C01810=1088.050,222.175,424.742,176.092,21.360,153.325
C01811=1088.041,221.787,424.782,176.088,21.356,153.325
C01812=1088.035,221.538,424.807,176.086,21.354,153.325
C01813=1088.029,221.290,424.832,176.082,21.351,153.325
C01814=1088.024,221.041,424.857,176.080,21.349,153.324
C01815=1088.018,220.792,424.883,176.077,21.347,153.324
C01816=1088.012,220.544,424.908,176.075,21.344,153.324
C01817=1088.007,220.295,424.932,176.072,21.341,153.324
C01818=1088.000,220.046,424.958,176.069,21.339,153.324
C01819=1087.995,219.798,424.983,176.066,21.336,153.324
C01820=1087.990,219.549,425.008,176.064,21.334,153.324
C01821=1087.984,219.301,425.033,176.061,21.332,153.324
C01822=1087.978,219.051,425.057,176.058,21.329,153.324
C01823=1087.973,218.803,425.083,176.055,21.327,153.324
C01824=1087.967,218.554,425.108,176.053,21.325,153.323
C01825=1087.961,218.305,425.133,176.050,21.322,153.323
C01826=1087.955,218.057,425.158,176.048,21.320,153.323
C01827=1087.950,217.808,425.182,176.044,21.317,153.323
C01828=1087.945,217.560,425.208,176.042,21.314,153.323
C01829=1087.939,217.310,425.233,176.039,21.312,153.323
C01830=1087.934,217.062,425.257,176.037,21.310,153.323
C01831=1087.927,216.813,425.282,176.035,21.307,153.323
C01832=1087.922,216.564,425.307,176.031,21.305,153.323
C01833=1087.917,216.315,425.332,176.029,21.303,153.322
C01834=1087.911,216.067,425.357,176.026,21.300,153.322
C01835=1087.905,215.818,425.382,176.024,21.298,153.322
C01836=1087.900,215.570,425.406,176.021,21.295,153.322
C01837=1087.894,215.320,425.431,176.018,21.292,153.322
C01838=1087.888,215.072,425.456,176.015,21.290,153.322
C01839=1087.883,214.824,425.480,176.013,21.288,153.322
C01840=1087.877,214.575,425.506,176.010,21.285,153.322
C01841=1087.872,214.326,425.530,176.008,21.283,153.322
C01842=1087.866,214.077,425.555,176.005,21.280,153.322
C01843=1087.861,213.829,425.580,176.002,21.278,153.321
C01844=1087.855,213.580,425.605,175.999,21.275,153.321
C01845=1087.849,213.331,425.629,175.997,21.273,153.321
C01846=1087.844,213.082,425.653,175.995,21.270,153.321
C01847=1087.838,212.834,425.678,175.991,21.268,153.321
C01848=1087.833,212.585,425.703,175.989,21.266,153.321
C01849=1087.827,212.336,425.727,175.986,21.263,153.321
C01850=1087.821,212.087,425.752,175.984,21.261,153.321
C01851=1087.815,211.839,425.777,175.981,21.258,153.321
C01852=1087.810,211.590,425.801,175.978,21.256,153.321
C01853=1087.805,211.341,425.825,175.975,21.253,153.320
C01854=1087.799,211.092,425.850,175.973,21.251,153.320
C01855=1087.793,210.844,425.874,175.970,21.248,153.320
C01856=1087.787,210.595,425.900,175.968,21.246,153.320
C01857=1087.782,210.346,425.924,175.965,21.244,153.320
C01858=1087.777,210.098,425.948,175.962,21.241,153.320
C01859=1087.771,209.848,425.973,175.960,21.239,153.320
C01860=1087.762,209.464,426.010,175.955,21.235,153.320
C01861=1087.754,209.080,426.048,175.952,21.231,153.319
C01862=1087.745,208.695,426.086,175.948,21.228,153.319
C01863=1087.736,208.311,426.123,175.944,21.224,153.319
C01864=1087.713,207.286,426.222,175.868,21.185,153.323
C01865=1087.707,207.037,426.246,175.866,21.184,153.323
C01866=1087.702,206.788,426.269,175.863,21.182,153.323
C01867=1087.696,206.539,426.293,175.860,21.181,153.323
C01868=1087.690,206.291,426.318,175.857,21.179,153.323
C01869=1087.685,206.042,426.342,175.855,21.178,153.323
C01870=1087.679,205.793,426.365,175.852,21.176,153.323
C01871=1087.674,205.545,426.389,175.849,21.175,153.324
C01872=1087.669,205.296,426.413,175.846,21.173,153.324
C01873=1087.662,205.046,426.437,175.843,21.172,153.324
C01874=1087.657,204.798,426.461,175.841,21.170,153.324
C01875=1087.651,204.549,426.484,175.838,21.169,153.324
C01876=1087.646,204.300,426.508,175.836,21.167,153.324
C01877=1087.641,204.052,426.532,175.833,21.166,153.324
C01878=1087.635,203.803,426.555,175.829,21.164,153.324
C01879=1087.630,203.554,426.580,175.827,21.163,153.325
C01880=1087.624,203.305,426.603,175.824,21.161,153.325
C01881=1087.618,203.056,426.627,175.822,21.159,153.325
C01882=1087.613,202.807,426.651,175.819,21.158,153.325
C01883=1087.607,202.559,426.674,175.817,21.156,153.325
C01884=1087.601,202.310,426.697,175.814,21.155,153.325
C01885=1087.596,202.061,426.722,175.811,21.153,153.325
C01886=1087.590,201.812,426.744,175.808,21.152,153.325
C01887=1087.585,201.564,426.769,175.805,21.151,153.325
C01888=1087.579,201.314,426.792,175.803,21.149,153.326
C01889=1087.573,201.066,426.816,175.800,21.148,153.326
C01890=1087.568,200.816,426.839,175.797,21.147,153.326
C01891=1087.562,200.568,426.863,175.795,21.145,153.326
C01892=1087.556,200.319,426.886,175.791,21.143,153.326
C01893=1087.550,200.071,426.910,175.789,21.142,153.326
C01894=1087.545,199.822,426.933,175.786,21.140,153.326
C01895=1087.539,199.573,426.956,175.784,21.139,153.326
C01896=1087.533,199.324,426.981,175.781,21.138,153.326
C01897=1087.527,199.075,427.004,175.778,21.136,153.327
C01898=1087.522,198.826,427.027,175.776,21.135,153.327
C01899=1087.516,198.577,427.051,175.773,21.133,153.327
C01900=1087.511,198.328,427.074,175.770,21.131,153.327
C01901=1087.505,198.079,427.097,175.767,21.130,153.327
C01902=1087.500,197.831,427.121,175.764,21.129,153.327
C01903=1087.494,197.582,427.144,175.762,21.127,153.327
C01904=1087.488,197.333,427.167,175.759,21.125,153.327
C01905=1087.483,197.084,427.191,175.757,21.124,153.327
C01906=1087.477,196.836,427.214,175.754,21.122,153.327
C01907=1087.471,196.587,427.237,175.752,21.121,153.328
C01908=1087.466,196.337,427.260,175.749,21.120,153.328
C01909=1087.460,196.089,427.284,175.746,21.118,153.328
C01910=1087.455,195.840,427.307,175.743,21.116,153.328
C01911=1087.449,195.591,427.330,175.740,21.115,153.328
C01912=1087.444,195.342,427.354,175.738,21.113,153.328
C01913=1087.438,195.093,427.377,175.735,21.112,153.328
C01914=1087.432,194.845,427.400,175.733,21.111,153.328
C01915=1087.426,194.596,427.423,175.730,21.109,153.329
C01916=1087.421,194.347,427.447,175.727,21.108,153.329
C01917=1087.416,194.098,427.470,175.725,21.106,153.329
C01918=1087.410,193.849,427.493,175.722,21.104,153.329
C01919=1087.404,193.600,427.516,175.720,21.103,153.329
C01920=1087.399,193.351,427.539,175.716,21.101,153.329
C01921=1087.393,193.103,427.563,175.714,21.100,153.329
C01922=1087.387,192.854,427.586,175.711,21.098,153.329
C01923=1087.382,192.605,427.609,175.709,21.097,153.329
C01924=1087.376,192.356,427.632,175.706,21.095,153.329
C01925=1087.371,192.079,427.657,175.703,21.094,153.330
C01926=1087.364,191.801,427.683,175.700,21.092,153.330
C01927=1087.358,191.523,427.709,175.697,21.090,153.330
C01928=1087.352,191.245,427.734,175.694,21.088,153.330
C01929=1087.347,190.997,427.757,175.691,21.087,153.330
C01930=1087.341,190.748,427.780,175.689,21.085,153.330
C01931=1087.336,190.499,427.804,175.686,21.084,153.330
C01932=1087.330,190.250,427.826,175.684,21.082,153.330
C01933=1087.324,190.001,427.849,175.681,21.081,153.330
C01934=1087.319,189.752,427.872,175.679,21.079,153.330
C01935=1087.313,189.503,427.895,175.676,21.078,153.331
C01936=1087.307,189.254,427.918,175.673,21.076,153.331
C01937=1087.303,189.006,427.941,175.671,21.075,153.331
C01938=1087.297,188.757,427.964,175.668,21.073,153.331
C01939=1087.291,188.508,427.987,175.666,21.072,153.331
C01940=1087.286,188.259,428.010,175.663,21.070,153.331
C01941=1087.280,188.010,428.032,175.661,21.069,153.331
C01942=1087.275,187.761,428.055,175.658,21.067,153.331
C01943=1087.269,187.513,428.078,175.656,21.066,153.331
C01944=1087.264,187.263,428.102,175.653,21.064,153.331
C01945=1087.259,187.014,428.125,175.650,21.063,153.331
C01946=1087.253,186.766,428.147,175.648,21.061,153.332
C01947=1087.248,186.517,428.169,175.645,21.059,153.332
C01948=1087.242,186.268,428.192,175.642,21.057,153.332
C01949=1087.237,186.019,428.215,175.639,21.056,153.332
C01950=1087.231,185.770,428.238,175.637,21.055,153.332
C01951=1087.226,185.522,428.261,175.634,21.053,153.332
C01952=1087.220,185.272,428.283,175.632,21.051,153.332
C01953=1087.215,185.023,428.307,175.629,21.050,153.332
C01954=1087.209,184.775,428.329,175.627,21.048,153.332
C01955=1087.203,184.525,428.351,175.624,21.047,153.332
C01956=1087.198,184.276,428.374,175.621,21.046,153.332
C01957=1087.192,184.027,428.397,175.619,21.044,153.333
C01958=1087.186,183.779,428.419,175.616,21.043,153.333
C01959=1087.181,183.530,428.441,175.614,21.041,153.333
C01960=1087.175,183.281,428.464,175.611,21.040,153.333
C01961=1087.169,183.032,428.487,175.609,21.038,153.333
C01962=1087.163,182.783,428.509,175.606,21.037,153.333
C01963=1087.157,182.534,428.532,175.603,21.035,153.333
C01964=1087.152,182.286,428.554,175.601,21.034,153.333
C01965=1087.147,182.036,428.576,175.598,21.032,153.333
C01966=1087.140,181.788,428.599,175.596,21.031,153.333
C01967=1087.135,181.538,428.621,175.593,21.030,153.334
C01968=1087.129,181.289,428.644,175.590,21.028,153.334
C01969=1087.123,181.041,428.666,175.588,21.027,153.334
C01970=1087.118,180.792,428.688,175.585,21.025,153.334
C01971=1087.112,180.543,428.711,175.583,21.024,153.334
C01972=1087.107,180.293,428.733,175.580,21.022,153.334
C01973=1087.100,180.045,428.756,175.578,21.021,153.334
C01974=1087.095,179.796,428.778,175.575,21.019,153.334
C01975=1087.090,179.547,428.801,175.572,21.018,153.334
C01976=1087.083,179.298,428.822,175.570,21.016,153.335
C01977=1087.078,179.049,428.845,175.567,21.015,153.335
C01978=1087.073,178.800,428.867,175.565,21.013,153.335
C01979=1087.066,178.552,428.889,175.562,21.012,153.335
C01980=1087.061,178.302,428.912,175.560,21.011,153.335
C01981=1087.055,178.053,428.935,175.558,21.009,153.335
C01982=1087.050,177.805,428.956,175.555,21.008,153.335
C01983=1087.044,177.555,428.978,175.553,21.006,153.335
C01984=1087.039,177.306,429.001,175.550,21.005,153.335
C01985=1087.033,177.058,429.022,175.548,21.003,153.335
C01986=1087.027,176.809,429.045,175.545,21.002,153.335
C01987=1087.021,176.560,429.067,175.543,21.000,153.335
C01988=1087.016,176.310,429.089,175.540,20.999,153.336
C01989=1087.010,176.033,429.114,175.537,20.996,153.336
C01990=1087.003,175.755,429.139,175.534,20.995,153.336
C01991=1086.997,175.476,429.164,175.531,20.994,153.336
C01992=1086.991,175.199,429.188,175.529,20.992,153.336
C01993=1086.985,174.949,429.210,175.526,20.991,153.336
C01994=1086.980,174.701,429.232,175.524,20.989,153.336
C01995=1086.974,174.452,429.254,175.521,20.987,153.336
C01996=1086.969,174.203,429.276,175.519,20.986,153.336
C01997=1086.963,173.955,429.298,175.516,20.984,153.336
C01998=1086.957,173.705,429.321,175.514,20.983,153.336
C01999=1086.952,173.456,429.343,175.511,20.981,153.337
C02000=1086.946,173.207,429.364,175.508,20.980,153.337
C02001=1086.941,172.958,429.387,175.506,20.978,153.337
C02002=1086.935,172.710,429.408,175.504,20.976,153.337
C02003=1086.930,172.460,429.430,175.501,20.975,153.337
C02004=1086.923,172.211,429.452,175.498,20.974,153.337
C02005=1086.919,171.962,429.474,175.496,20.972,153.337
C02006=1086.913,171.713,429.497,175.493,20.970,153.337
C02007=1086.907,171.465,429.518,175.491,20.969,153.337
C02008=1086.902,171.215,429.540,175.489,20.967,153.337
C02009=1086.896,170.967,429.562,175.487,20.966,153.337
C02010=1086.891,170.717,429.584,175.484,20.965,153.337
C02011=1086.885,170.468,429.606,175.482,20.963,153.337
C02012=1086.880,170.219,429.627,175.479,20.961,153.337
C02013=1086.874,169.970,429.649,175.476,20.960,153.338
C02014=1086.869,169.722,429.672,175.474,20.958,153.338
C02015=1086.862,169.473,429.693,175.471,20.956,153.338
C02016=1086.858,169.224,429.715,175.469,20.955,153.338
C02017=1086.851,168.975,429.737,175.466,20.953,153.338
C02018=1086.847,168.726,429.759,175.464,20.952,153.338
C02019=1086.840,168.477,429.780,175.461,20.950,153.338
C02020=1086.836,168.228,429.802,175.460,20.949,153.338
C02021=1086.829,167.979,429.824,175.457,20.947,153.338
C02022=1086.825,167.730,429.846,175.455,20.945,153.338
C02023=1086.818,167.481,429.867,175.452,20.944,153.338
C02024=1086.814,167.232,429.889,175.450,20.942,153.338
C02025=1086.807,166.983,429.911,175.447,20.941,153.338
C02026=1086.803,166.734,429.933,175.445,20.939,153.338
C02027=1086.796,166.485,429.954,175.442,20.937,153.338
C02028=1086.792,166.236,429.976,175.440,20.936,153.339
C02029=1086.786,165.987,429.997,175.437,20.934,153.339
C02030=1086.781,165.738,430.020,175.435,20.933,153.339
C02031=1086.775,165.489,430.041,175.433,20.931,153.339
C02032=1086.770,165.239,430.062,175.431,20.930,153.339
C02033=1086.764,164.991,430.084,175.428,20.928,153.339
C02034=1086.758,164.741,430.105,175.426,20.926,153.339
C02035=1086.753,164.493,430.127,175.423,20.925,153.339
C02036=1086.748,164.244,430.148,175.421,20.923,153.339
C02037=1086.742,163.994,430.171,175.418,20.921,153.339
C02038=1086.737,163.746,430.192,175.416,20.920,153.339
C02039=1086.732,163.496,430.213,175.413,20.918,153.339
C02040=1086.726,163.247,430.235,175.411,20.917,153.339
C02041=1086.721,162.999,430.256,175.409,20.915,153.339
C02042=1086.715,162.749,430.278,175.406,20.914,153.339
C02043=1086.710,162.501,430.300,175.404,20.912,153.339
C02044=1086.705,162.251,430.321,175.402,20.910,153.339
C02045=1086.699,162.002,430.342,175.399,20.908,153.339
C02046=1086.693,161.754,430.364,175.397,20.907,153.339
C02047=1086.689,161.505,430.385,175.394,20.905,153.339
C02048=1086.683,161.255,430.406,175.392,20.904,153.339
C02049=1086.677,161.007,430.428,175.390,20.903,153.340
C02050=1086.671,160.757,430.449,175.387,20.901,153.340
C02051=1086.665,160.509,430.471,175.385,20.899,153.340
C02052=1086.660,160.259,430.492,175.382,20.897,153.340
C02053=1086.654,159.981,430.516,175.380,20.896,153.340
C02054=1086.647,159.703,430.539,175.377,20.894,153.340
C02055=1086.642,159.424,430.563,175.375,20.893,153.340
C02056=1086.635,159.146,430.587,175.372,20.890,153.340
C02057=1086.630,158.897,430.608,175.370,20.889,153.340
C02058=1086.623,158.648,430.629,175.367,20.888,153.340
C02059=1086.618,158.399,430.650,175.365,20.886,153.340
C02060=1086.613,158.150,430.672,175.362,20.884,153.340
C02061=1086.607,157.901,430.694,175.360,20.883,153.340
C02062=1086.602,157.652,430.714,175.357,20.881,153.340
C02063=1086.596,157.403,430.735,175.355,20.879,153.340
C02064=1086.590,157.153,430.756,175.353,20.878,153.340
C02065=1086.585,156.905,430.778,175.351,20.876,153.340
C02066=1086.580,156.656,430.798,175.348,20.875,153.341
C02067=1086.573,156.407,430.820,175.346,20.873,153.341
C02068=1086.568,156.158,430.841,175.343,20.872,153.341
C02069=1086.563,155.909,430.862,175.341,20.870,153.341
C02070=1086.556,155.660,430.883,175.339,20.869,153.341
C02071=1086.551,155.411,430.904,175.337,20.867,153.341
C02072=1086.546,155.162,430.925,175.334,20.865,153.341
C02073=1086.540,154.912,430.946,175.332,20.863,153.341
C02074=1086.534,154.664,430.967,175.329,20.862,153.341
C02075=1086.529,154.415,430.988,175.327,20.861,153.341
C02076=1086.523,154.165,431.009,175.325,20.859,153.341
C02077=1086.518,153.916,431.030,175.323,20.858,153.341
C02078=1086.512,153.667,431.051,175.320,20.856,153.341
C02079=1086.506,153.418,431.072,175.318,20.854,153.341
C02080=1086.501,153.169,431.093,175.315,20.852,153.341
C02081=1086.495,152.920,431.114,175.314,20.851,153.341
C02082=1086.489,152.670,431.135,175.311,20.850,153.341
C02083=1086.484,152.421,431.155,175.309,20.848,153.341
C02084=1086.479,152.173,431.177,175.306,20.846,153.341
C02085=1086.473,151.924,431.197,175.304,20.844,153.341
C02086=1086.468,151.674,431.218,175.302,20.843,153.341
C02087=1086.462,151.425,431.239,175.300,20.841,153.341
C02088=1086.457,151.176,431.260,175.297,20.840,153.342
C02089=1086.451,150.927,431.281,175.295,20.838,153.342
C02090=1086.445,150.678,431.302,175.292,20.837,153.342
C02091=1086.439,150.429,431.322,175.290,20.835,153.342
C02092=1086.434,150.180,431.343,175.288,20.833,153.342
C02093=1086.429,149.932,431.364,175.286,20.832,153.342
C02094=1086.423,149.682,431.385,175.283,20.830,153.342
C02095=1086.417,149.433,431.405,175.281,20.829,153.342
C02096=1086.412,149.183,431.426,175.278,20.827,153.342
C02097=1086.406,148.935,431.447,175.277,20.825,153.342
C02098=1086.401,148.686,431.467,175.274,20.824,153.342
C02099=1086.395,148.436,431.488,175.272,20.822,153.342
C02100=1086.389,148.187,431.509,175.269,20.820,153.342
C02101=1086.384,147.939,431.530,175.268,20.819,153.342
C02102=1086.378,147.690,431.550,175.265,20.818,153.342
C02103=1086.372,147.440,431.571,175.263,20.816,153.342
C02104=1086.367,147.191,431.591,175.260,20.814,153.342
C02105=1086.362,146.942,431.612,175.258,20.812,153.342
C02106=1086.355,146.694,431.633,175.256,20.811,153.342
C02107=1086.350,146.444,431.653,175.253,20.809,153.342
C02108=1086.344,146.195,431.674,175.251,20.807,153.342
C02109=1086.339,145.946,431.695,175.249,20.806,153.342
C02110=1086.333,145.697,431.715,175.247,20.805,153.342
C02111=1086.328,145.448,431.735,175.245,20.803,153.342
C02112=1086.322,145.198,431.756,175.242,20.801,153.342
C02113=1086.316,144.949,431.776,175.240,20.799,153.342
C02114=1086.311,144.700,431.797,175.237,20.797,153.342
C02115=1086.305,144.451,431.817,175.236,20.796,153.342
C02116=1086.299,144.203,431.838,175.233,20.795,153.342
C02117=1086.293,143.924,431.860,175.231,20.793,153.342
C02118=1086.286,143.645,431.884,175.228,20.791,153.343
C02119=1086.281,143.367,431.906,175.226,20.789,153.343
C02120=1086.274,143.087,431.929,175.223,20.787,153.343
C02121=1086.269,142.838,431.949,175.221,20.786,153.343
C02122=1086.263,142.589,431.969,175.218,20.784,153.343
C02123=1086.258,142.340,431.990,175.216,20.782,153.343
C02124=1086.252,142.091,432.011,175.214,20.781,153.343
C02125=1086.246,141.842,432.031,175.212,20.779,153.343
C02126=1086.241,141.593,432.051,175.210,20.777,153.343
C02127=1086.236,141.344,432.072,175.207,20.775,153.343
C02128=1086.230,141.095,432.092,175.205,20.774,153.343
C02129=1086.225,140.846,432.112,175.203,20.772,153.343
C02130=1086.219,140.596,432.133,175.201,20.771,153.343
C02131=1086.213,140.347,432.153,175.198,20.769,153.343
C02132=1086.208,140.098,432.174,175.197,20.768,153.343
C02133=1086.202,139.850,432.194,175.194,20.766,153.343
C02134=1086.196,139.600,432.214,175.192,20.764,153.343
C02135=1086.190,139.352,432.234,175.189,20.762,153.343
C02136=1086.185,139.102,432.254,175.188,20.761,153.343
C02137=1086.179,138.853,432.274,175.185,20.759,153.343
C02138=1086.174,138.604,432.294,175.183,20.758,153.343
C02139=1086.168,138.355,432.314,175.180,20.756,153.343
C02140=1086.163,138.106,432.335,175.179,20.754,153.343
C02141=1086.157,137.857,432.355,175.176,20.753,153.343
C02142=1086.151,137.607,432.375,175.174,20.751,153.343
C02143=1086.145,137.358,432.395,175.172,20.749,153.343
C02144=1086.140,137.109,432.416,175.170,20.747,153.343
C02145=1086.134,136.860,432.436,175.167,20.746,153.343
C02146=1086.128,136.611,432.455,175.165,20.744,153.343
C02147=1086.123,136.361,432.475,175.163,20.742,153.343
C02148=1086.117,136.113,432.495,175.161,20.741,153.343
C02149=1086.112,135.863,432.516,175.159,20.739,153.343
C02150=1086.106,135.614,432.535,175.156,20.737,153.343
C02151=1086.101,135.365,432.556,175.155,20.736,153.343
C02152=1086.095,135.116,432.576,175.152,20.734,153.343
C02153=1086.089,134.867,432.596,175.150,20.733,153.343
C02154=1086.084,134.618,432.615,175.147,20.731,153.343
C02155=1086.078,134.369,432.635,175.146,20.729,153.343
C02156=1086.073,134.120,432.656,175.143,20.727,153.343
C02157=1086.067,133.870,432.675,175.141,20.725,153.343
C02158=1086.061,133.621,432.695,175.139,20.724,153.343
C02159=1086.056,133.372,432.716,175.137,20.722,153.343
C02160=1086.050,133.123,432.735,175.135,20.721,153.343
C02161=1086.045,132.874,432.755,175.132,20.719,153.343
C02162=1086.039,132.624,432.775,175.131,20.717,153.343
C02163=1086.033,132.375,432.795,175.128,20.716,153.343
C02164=1086.028,132.126,432.815,175.126,20.714,153.343
C02165=1086.022,131.877,432.834,175.124,20.712,153.343
C02166=1086.016,131.628,432.854,175.122,20.710,153.343
C02167=1086.011,131.379,432.874,175.119,20.709,153.343
C02168=1086.005,131.130,432.894,175.118,20.708,153.343
C02169=1086.000,130.880,432.913,175.115,20.706,153.343
C02170=1085.994,130.631,432.933,175.113,20.704,153.343
C02171=1085.988,130.382,432.953,175.110,20.702,153.343
C02172=1085.982,130.133,432.973,175.109,20.701,153.343
C02173=1085.976,129.884,432.992,175.107,20.699,153.343
C02174=1085.970,129.635,433.012,175.104,20.697,153.343
C02175=1085.965,129.385,433.032,175.103,20.695,153.343
C02176=1085.959,129.136,433.052,175.100,20.694,153.343
C02177=1085.954,128.887,433.071,175.098,20.692,153.343
C02178=1085.948,128.638,433.091,175.096,20.691,153.343
C02179=1085.942,128.389,433.110,175.094,20.689,153.343
C02180=1085.937,128.140,433.130,175.091,20.687,153.343
C02181=1085.930,127.861,433.152,175.089,20.685,153.343
C02182=1085.924,127.582,433.174,175.087,20.683,153.343
C02183=1085.917,127.304,433.195,175.084,20.682,153.343
C02184=1085.912,127.025,433.218,175.082,20.680,153.343
C02185=1085.906,126.776,433.237,175.080,20.678,153.343
C02186=1085.900,126.527,433.257,175.078,20.676,153.343
C02187=1085.894,126.278,433.276,175.075,20.674,153.343
C02188=1085.889,126.028,433.295,175.074,20.673,153.343
C02189=1085.883,125.779,433.315,175.072,20.671,153.343
C02190=1085.877,125.530,433.335,175.069,20.669,153.343
C02191=1085.872,125.281,433.354,175.068,20.668,153.343
C02192=1085.866,125.032,433.374,175.065,20.666,153.343
C02193=1085.861,124.783,433.393,175.063,20.664,153.343
C02194=1085.855,124.533,433.413,175.061,20.663,153.343
C02195=1085.849,124.284,433.433,175.059,20.661,153.343
C02196=1085.843,124.035,433.452,175.056,20.659,153.343
C02197=1085.838,123.786,433.471,175.055,20.657,153.343
C02198=1085.833,123.537,433.490,175.053,20.655,153.343
C02199=1085.827,123.288,433.510,175.050,20.654,153.343
C02200=1085.821,123.039,433.529,175.049,20.652,153.343
C02201=1085.815,122.789,433.548,175.046,20.650,153.343
C02202=1085.810,122.540,433.568,175.044,20.648,153.343
C02203=1085.804,122.291,433.588,175.042,20.647,153.343
C02204=1085.799,122.042,433.606,175.040,20.645,153.343
C02205=1085.793,121.793,433.626,175.038,20.643,153.343
C02206=1085.787,121.543,433.645,175.036,20.641,153.343
C02207=1085.781,121.294,433.664,175.034,20.639,153.343
C02208=1085.775,121.045,433.684,175.031,20.638,153.343
C02209=1085.771,120.796,433.704,175.030,20.636,153.343
C02210=1085.765,120.547,433.723,175.028,20.634,153.343
C02211=1085.760,120.297,433.742,175.025,20.632,153.343
C02212=1085.754,120.048,433.761,175.024,20.631,153.343
C02213=1085.748,119.798,433.781,175.021,20.629,153.343
C02214=1085.743,119.550,433.799,175.019,20.627,153.343
C02215=1085.737,119.301,433.819,175.017,20.625,153.343
C02216=1085.732,119.051,433.839,175.015,20.624,153.343
C02217=1085.726,118.802,433.858,175.014,20.622,153.343
C02218=1085.721,118.553,433.877,175.011,20.620,153.343
C02219=1085.715,118.304,433.896,175.009,20.618,153.343
C02220=1085.709,118.054,433.915,175.007,20.617,153.343
C02221=1085.704,117.806,433.934,175.005,20.615,153.343
C02222=1085.699,117.556,433.953,175.003,20.613,153.343
C02223=1085.693,117.307,433.973,175.001,20.611,153.343
C02224=1085.687,117.057,433.992,174.999,20.609,153.343
C02225=1085.681,116.809,434.010,174.996,20.608,153.343
C02226=1085.676,116.559,434.029,174.995,20.606,153.342
C02227=1085.670,116.310,434.049,174.993,20.604,153.342
C02228=1085.665,116.061,434.067,174.991,20.602,153.342
C02229=1085.659,115.812,434.087,174.989,20.600,153.342
C02230=1085.654,115.562,434.106,174.986,20.598,153.342
C02231=1085.649,115.314,434.125,174.985,20.597,153.342
C02232=1085.643,115.064,434.144,174.983,20.595,153.342
C02233=1085.637,114.815,434.163,174.980,20.593,153.342
C02234=1085.632,114.566,434.182,174.979,20.591,153.342
C02235=1085.626,114.317,434.201,174.977,20.589,153.342
C02236=1085.621,114.067,434.221,174.975,20.588,153.342
C02237=1085.614,113.818,434.239,174.973,20.586,153.342
C02238=1085.609,113.569,434.258,174.970,20.584,153.342
C02239=1085.604,113.319,434.277,174.969,20.582,153.342
C02240=1085.598,113.070,434.296,174.966,20.580,153.342
C02241=1085.593,112.821,434.315,174.964,20.578,153.342
C02242=1085.587,112.572,434.334,174.963,20.577,153.342
C02243=1085.581,112.323,434.353,174.960,20.575,153.342
C02244=1085.576,112.074,434.372,174.959,20.574,153.342
C02245=1085.570,111.795,434.393,174.957,20.571,153.342
C02246=1085.563,111.516,434.414,174.954,20.569,153.342
C02247=1085.556,111.237,434.434,174.952,20.567,153.342
C02248=1085.550,110.958,434.455,174.949,20.565,153.342
C02249=1085.545,110.710,434.474,174.947,20.563,153.342
C02250=1085.539,110.461,434.493,174.946,20.561,153.342
C02251=1085.533,110.211,434.512,174.943,20.559,153.342
C02252=1085.528,109.961,434.531,174.942,20.558,153.341
C02253=1085.522,109.713,434.549,174.940,20.556,153.341
C02254=1085.516,109.463,434.568,174.937,20.554,153.341
C02255=1085.511,109.215,434.587,174.936,20.553,153.341
C02256=1085.505,108.965,434.605,174.933,20.551,153.341
C02257=1085.499,108.715,434.624,174.932,20.549,153.341
C02258=1085.493,108.467,434.643,174.929,20.547,153.341
C02259=1085.488,108.217,434.661,174.927,20.545,153.341
C02260=1085.482,107.967,434.680,174.926,20.543,153.341
C02261=1085.476,107.719,434.699,174.923,20.541,153.341
C02262=1085.471,107.469,434.717,174.922,20.540,153.341
C02263=1085.465,107.220,434.736,174.919,20.538,153.341
C02264=1085.460,106.971,434.755,174.917,20.536,153.341
C02265=1085.454,106.721,434.773,174.916,20.534,153.341
C02266=1085.448,106.473,434.792,174.913,20.532,153.341
C02267=1085.443,106.223,434.811,174.912,20.531,153.341
C02268=1085.436,105.973,434.829,174.910,20.529,153.341
C02269=1085.431,105.725,434.848,174.907,20.527,153.341
C02270=1085.425,105.476,434.866,174.906,20.525,153.341
C02271=1085.420,105.226,434.884,174.904,20.523,153.341
C02272=1085.415,104.977,434.904,174.902,20.522,153.341
C02273=1085.409,104.728,434.921,174.900,20.520,153.341
C02274=1085.403,104.478,434.940,174.898,20.518,153.341
C02275=1085.398,104.229,434.958,174.896,20.516,153.340
C02276=1085.392,103.980,434.977,174.894,20.514,153.340
C02277=1085.386,103.731,434.996,174.892,20.512,153.340
C02278=1085.381,103.481,435.014,174.890,20.510,153.340
C02279=1085.374,103.232,435.033,174.889,20.508,153.340
C02280=1085.370,102.983,435.051,174.886,20.506,153.340
C02281=1085.363,102.734,435.070,174.885,20.505,153.340
C02282=1085.358,102.484,435.088,174.882,20.503,153.340
C02283=1085.353,102.235,435.107,174.880,20.501,153.340
C02284=1085.347,101.986,435.124,174.879,20.499,153.340
C02285=1085.342,101.736,435.143,174.876,20.497,153.340
C02286=1085.336,101.488,435.161,174.875,20.495,153.340
C02287=1085.331,101.237,435.180,174.873,20.493,153.340
C02288=1085.325,100.989,435.198,174.871,20.492,153.340
C02289=1085.319,100.739,435.216,174.869,20.490,153.340
C02290=1085.314,100.491,435.235,174.866,20.488,153.340
C02291=1085.308,100.241,435.253,174.865,20.486,153.339
C02292=1085.302,99.992,435.271,174.863,20.484,153.339
C02293=1085.296,99.742,435.290,174.861,20.483,153.339
C02294=1085.291,99.493,435.307,174.859,20.481,153.339
C02295=1085.284,99.244,435.326,174.858,20.479,153.339
C02296=1085.280,98.995,435.344,174.855,20.477,153.339
C02297=1085.273,98.745,435.362,174.854,20.475,153.339
C02298=1085.268,98.497,435.380,174.851,20.473,153.339
C02299=1085.262,98.247,435.399,174.849,20.471,153.339
C02300=1085.257,97.998,435.416,174.848,20.469,153.339
C02301=1085.250,97.748,435.435,174.845,20.467,153.339
C02302=1085.246,97.499,435.453,174.844,20.465,153.339
C02303=1085.239,97.249,435.471,174.842,20.464,153.339
C02304=1085.234,97.001,435.489,174.840,20.462,153.339
C02305=1085.227,96.751,435.507,174.838,20.460,153.339
C02306=1085.223,96.502,435.525,174.837,20.458,153.339
C02307=1085.216,96.253,435.544,174.834,20.456,153.339
C02308=1085.211,96.004,435.562,174.832,20.454,153.339
C02309=1085.205,95.724,435.582,174.831,20.452,153.338
C02310=1085.198,95.446,435.602,174.828,20.450,153.338
C02311=1085.191,95.168,435.623,174.826,20.448,153.338
C02312=1085.186,94.889,435.643,174.824,20.446,153.338
C02313=1085.180,94.639,435.661,174.822,20.444,153.338
C02314=1085.174,94.390,435.678,174.820,20.442,153.338
C02315=1085.169,94.142,435.697,174.819,20.441,153.338
C02316=1085.163,93.892,435.715,174.816,20.438,153.338
C02317=1085.158,93.643,435.733,174.814,20.436,153.338
C02318=1085.152,93.393,435.751,174.813,20.434,153.338
C02319=1085.146,93.144,435.768,174.810,20.432,153.338
C02320=1085.141,92.895,435.787,174.809,20.431,153.338
C02321=1085.135,92.645,435.805,174.807,20.428,153.337
C02322=1085.129,92.396,435.822,174.805,20.427,153.337
C02323=1085.123,92.147,435.840,174.803,20.424,153.337
C02324=1085.118,91.897,435.859,174.802,20.423,153.337
C02325=1085.113,91.648,435.876,174.799,20.421,153.337
C02326=1085.107,91.398,435.894,174.798,20.419,153.337
C02327=1085.101,91.149,435.912,174.796,20.417,153.337
C02328=1085.096,90.900,435.929,174.794,20.415,153.337
C02329=1085.089,90.651,435.948,174.792,20.413,153.337
C02330=1085.085,90.402,435.966,174.790,20.412,153.337
C02331=1085.078,90.152,435.984,174.788,20.409,153.337
C02332=1085.073,89.903,436.002,174.786,20.407,153.337
C02333=1085.067,89.654,436.019,174.784,20.406,153.337
C02334=1085.061,89.404,436.037,174.782,20.403,153.336
C02335=1085.056,89.155,436.055,174.781,20.402,153.336
C02336=1085.050,88.905,436.073,174.778,20.400,153.336
C02337=1085.044,88.656,436.090,174.777,20.398,153.336
C02338=1085.039,88.407,436.108,174.775,20.396,153.336
C02339=1085.033,88.158,436.126,174.774,20.394,153.336
C02340=1085.027,87.909,436.143,174.771,20.392,153.336
C02341=1085.021,87.660,436.161,174.770,20.391,153.336
C02342=1085.015,87.410,436.179,174.768,20.388,153.336
C02343=1085.010,87.161,436.196,174.766,20.387,153.336
C02344=1085.004,86.912,436.214,174.764,20.384,153.336
C02345=1084.998,86.662,436.232,174.762,20.383,153.336
C02346=1084.993,86.413,436.249,174.760,20.381,153.336
C02347=1084.987,86.163,436.266,174.759,20.379,153.335
C02348=1084.981,85.914,436.284,174.756,20.377,153.335
C02349=1084.976,85.665,436.302,174.755,20.375,153.335
C02350=1084.970,85.416,436.319,174.753,20.373,153.335
C02351=1084.964,85.166,436.337,174.752,20.371,153.335
C02352=1084.959,84.917,436.355,174.749,20.369,153.335
C02353=1084.953,84.668,436.372,174.748,20.367,153.335
C02354=1084.947,84.418,436.390,174.746,20.365,153.335
C02355=1084.942,84.168,436.407,174.744,20.363,153.335
C02356=1084.936,83.919,436.425,174.742,20.361,153.335
C02357=1084.931,83.670,436.442,174.741,20.359,153.334
C02358=1084.925,83.420,436.460,174.738,20.357,153.334
C02359=1084.918,83.172,436.477,174.737,20.356,153.334
C02360=1084.913,82.923,436.495,174.735,20.353,153.334
C02361=1084.908,82.673,436.512,174.733,20.352,153.334
C02362=1084.902,82.423,436.529,174.731,20.349,153.334
C02363=1084.896,82.174,436.547,174.730,20.347,153.334
C02364=1084.891,81.925,436.565,174.727,20.345,153.334
C02365=1084.885,81.676,436.582,174.726,20.343,153.334
C02366=1084.879,81.426,436.599,174.724,20.342,153.334
C02367=1084.874,81.177,436.617,174.722,20.340,153.334
C02368=1084.868,80.928,436.634,174.720,20.338,153.334
C02369=1084.863,80.678,436.651,174.719,20.336,153.333
C02370=1084.857,80.429,436.669,174.716,20.334,153.333
C02371=1084.851,80.179,436.687,174.715,20.332,153.333
C02372=1084.845,79.931,436.704,174.713,20.330,153.333
C02373=1084.839,79.652,436.723,174.712,20.328,153.333
C02374=1084.833,79.374,436.743,174.709,20.325,153.333
C02375=1084.827,79.095,436.762,174.707,20.323,153.333
C02376=1084.821,78.816,436.782,174.705,20.321,153.333
C02377=1084.815,78.566,436.799,174.704,20.319,153.333
C02378=1084.809,78.317,436.816,174.701,20.317,153.333
C02379=1084.803,78.068,436.833,174.700,20.315,153.332
C02380=1084.798,77.819,436.850,174.698,20.313,153.332
C02381=1084.792,77.570,436.868,174.696,20.311,153.332
C02382=1084.786,77.320,436.884,174.694,20.309,153.332
C02383=1084.780,77.071,436.902,174.693,20.307,153.332
C02384=1084.775,76.822,436.919,174.691,20.305,153.332
C02385=1084.770,76.572,436.936,174.689,20.303,153.332
C02386=1084.763,76.322,436.954,174.688,20.301,153.332
C02387=1084.758,76.073,436.970,174.685,20.299,153.332
C02388=1084.752,75.824,436.988,174.684,20.297,153.331
C02389=1084.746,75.574,437.004,174.682,20.295,153.331
C02390=1084.741,75.325,437.022,174.681,20.293,153.331
C02391=1084.735,75.076,437.039,174.678,20.291,153.331
C02392=1084.729,74.826,437.057,174.677,20.289,153.331
C02393=1084.723,74.577,437.074,174.675,20.287,153.331
C02394=1084.718,74.328,437.090,174.673,20.285,153.331
C02395=1084.712,74.079,437.108,174.671,20.283,153.331
C02396=1084.706,73.829,437.124,174.670,20.282,153.331
C02397=1084.701,73.580,437.142,174.668,20.279,153.331
C02398=1084.696,73.330,437.159,174.666,20.277,153.330
C02399=1084.689,73.081,437.176,174.664,20.275,153.330
C02400=1084.683,72.831,437.193,174.663,20.273,153.330
C02401=1084.678,72.582,437.210,174.661,20.272,153.330
C02402=1084.672,72.333,437.227,174.659,20.269,153.330
C02403=1084.667,72.083,437.244,174.658,20.267,153.330
C02404=1084.661,71.835,437.261,174.655,20.265,153.330
C02405=1084.655,71.585,437.277,174.654,20.263,153.330
C02406=1084.650,71.336,437.295,174.652,20.261,153.330
C02407=1084.644,71.087,437.311,174.651,20.259,153.329
C02408=1084.638,70.836,437.328,174.648,20.257,153.329
C02409=1084.633,70.587,437.346,174.647,20.255,153.329
C02410=1084.627,70.338,437.362,174.645,20.253,153.329
C02411=1084.621,70.089,437.380,174.643,20.251,153.329
C02412=1084.615,69.839,437.396,174.642,20.249,153.329
C02413=1084.610,69.590,437.413,174.640,20.247,153.329
C02414=1084.604,69.341,437.430,174.638,20.246,153.329
C02415=1084.598,69.091,437.447,174.636,20.243,153.329
C02416=1084.592,68.842,437.463,174.635,20.241,153.328
C02417=1084.587,68.593,437.481,174.633,20.239,153.328
C02418=1084.581,68.344,437.497,174.631,20.237,153.328
C02419=1084.575,68.093,437.514,174.629,20.235,153.328
C02420=1084.569,67.845,437.531,174.628,20.233,153.328
C02421=1084.564,67.595,437.548,174.626,20.231,153.328
C02422=1084.558,67.346,437.564,174.624,20.229,153.328
C02423=1084.553,67.096,437.581,174.623,20.227,153.328
C02424=1084.546,66.847,437.598,174.621,20.225,153.328
C02425=1084.541,66.597,437.615,174.619,20.223,153.327
C02426=1084.535,66.348,437.631,174.617,20.221,153.327
C02427=1084.530,66.098,437.648,174.616,20.219,153.327
C02428=1084.524,65.850,437.665,174.613,20.217,153.327
C02429=1084.518,65.600,437.682,174.612,20.215,153.327
C02430=1084.512,65.351,437.698,174.611,20.213,153.327
C02431=1084.507,65.101,437.715,174.609,20.211,153.327
C02432=1084.501,64.852,437.731,174.607,20.209,153.327
C02433=1084.495,64.603,437.748,174.605,20.207,153.326
C02434=1084.490,64.353,437.765,174.604,20.205,153.326
C02435=1084.484,64.104,437.781,174.602,20.203,153.326
C02436=1084.478,63.855,437.797,174.600,20.201,153.326
C02437=1084.471,63.576,437.816,174.598,20.199,153.326
C02438=1084.465,63.297,437.835,174.597,20.197,153.326
C02439=1084.459,63.018,437.853,174.595,20.194,153.326
C02440=1084.452,62.740,437.872,174.592,20.192,153.326
C02441=1084.445,62.490,437.889,174.591,20.190,153.326
C02442=1084.440,62.241,437.905,174.589,20.188,153.325
C02443=1084.434,61.991,437.922,174.588,20.186,153.325
C02444=1084.428,61.742,437.938,174.585,20.184,153.325
C02445=1084.422,61.492,437.954,174.584,20.182,153.325
C02446=1084.416,61.243,437.970,174.582,20.180,153.325
C02447=1084.411,60.993,437.987,174.580,20.178,153.325
C02448=1084.405,60.744,438.004,174.579,20.176,153.325
C02449=1084.399,60.495,438.020,174.577,20.174,153.325
C02450=1084.393,60.245,438.036,174.575,20.172,153.325
C02451=1084.387,59.997,438.053,174.573,20.169,153.324
C02452=1084.382,59.747,438.070,174.572,20.168,153.324
C02453=1084.376,59.498,438.086,174.571,20.166,153.324
C02454=1084.370,59.248,438.102,174.568,20.164,153.324
C02455=1084.364,58.999,438.119,174.567,20.162,153.324
C02456=1084.358,58.750,438.135,174.565,20.160,153.324
C02457=1084.353,58.500,438.152,174.564,20.158,153.324
C02458=1084.347,58.251,438.168,174.562,20.156,153.324
C02459=1084.341,58.001,438.184,174.560,20.154,153.323
C02460=1084.335,57.751,438.200,174.559,20.152,153.323
C02461=1084.329,57.502,438.216,174.557,20.149,153.323
C02462=1084.325,57.253,438.233,174.555,20.148,153.323
C02463=1084.319,57.004,438.249,174.554,20.146,153.323
C02464=1084.313,56.754,438.265,174.552,20.143,153.323
C02465=1084.307,56.505,438.281,174.550,20.142,153.323
C02466=1084.301,56.256,438.298,174.548,20.139,153.323
C02467=1084.295,56.006,438.314,174.547,20.137,153.322
C02468=1084.290,55.757,438.331,174.545,20.135,153.322
C02469=1084.284,55.507,438.347,174.543,20.133,153.322
C02470=1084.278,55.258,438.363,174.542,20.131,153.322
C02471=1084.272,55.009,438.379,174.540,20.129,153.322
C02472=1084.266,54.759,438.395,174.538,20.127,153.322
C02473=1084.260,54.509,438.411,174.536,20.125,153.322
C02474=1084.255,54.261,438.427,174.535,20.123,153.322
C02475=1084.250,54.011,438.444,174.534,20.121,153.321
C02476=1084.244,53.762,438.460,174.531,20.118,153.321
C02477=1084.238,53.512,438.476,174.530,20.117,153.321
C02478=1084.232,53.262,438.492,174.528,20.114,153.321
C02479=1084.226,53.013,438.508,174.527,20.112,153.321
C02480=1084.220,52.764,438.525,174.525,20.111,153.321
C02481=1084.214,52.514,438.541,174.523,20.109,153.321
C02482=1084.209,52.266,438.557,174.522,20.107,153.321
C02483=1084.203,52.016,438.572,174.520,20.105,153.320
C02484=1084.198,51.766,438.589,174.518,20.102,153.320
C02485=1084.192,51.517,438.605,174.517,20.100,153.320
C02486=1084.186,51.267,438.622,174.515,20.098,153.320
C02487=1084.181,51.017,438.637,174.513,20.096,153.320
C02488=1084.175,50.769,438.653,174.512,20.094,153.320
C02489=1084.169,50.519,438.669,174.510,20.092,153.320
C02490=1084.164,50.269,438.685,174.509,20.090,153.319
C02491=1084.158,50.020,438.701,174.506,20.088,153.319
C02492=1084.152,49.771,438.717,174.505,20.086,153.319
C02493=1084.146,49.522,438.733,174.504,20.084,153.319
C02494=1084.141,49.272,438.749,174.502,20.081,153.319
C02495=1084.135,49.023,438.765,174.501,20.079,153.319
C02496=1084.130,48.773,438.782,174.498,20.077,153.319
C02497=1084.124,48.523,438.797,174.497,20.075,153.319
C02498=1084.119,48.274,438.813,174.496,20.073,153.318
C02499=1084.113,48.025,438.830,174.494,20.071,153.318
C02500=1084.107,47.775,438.845,174.492,20.069,153.318
C02501=1084.101,47.496,438.863,174.490,20.066,153.318
C02502=1084.094,47.217,438.881,174.489,20.064,153.318
C02503=1084.088,46.939,438.898,174.487,20.062,153.318
C02504=1084.082,46.660,438.916,174.485,20.059,153.317
C02505=1084.076,46.410,438.932,174.483,20.057,153.317
C02506=1084.070,46.161,438.948,174.481,20.055,153.317
C02507=1084.065,45.912,438.964,174.480,20.053,153.317
C02508=1084.059,45.662,438.980,174.479,20.051,153.317
C02509=1084.053,45.413,438.996,174.477,20.048,153.317
C02510=1084.048,45.163,439.011,174.475,20.046,153.316
C02511=1084.042,44.914,439.027,174.474,20.044,153.316
C02512=1084.037,44.664,439.043,174.472,20.042,153.316
C02513=1084.031,44.415,439.059,174.471,20.040,153.316
C02514=1084.026,44.165,439.074,174.468,20.038,153.316
C02515=1084.020,43.916,439.091,174.467,20.036,153.316
C02516=1084.014,43.666,439.106,174.466,20.034,153.316
C02517=1084.009,43.417,439.122,174.464,20.031,153.315
C02518=1084.002,43.168,439.137,174.463,20.029,153.315
C02519=1083.996,42.918,439.153,174.461,20.028,153.315
C02520=1083.991,42.668,439.169,174.459,20.026,153.315
C02521=1083.985,42.420,439.185,174.458,20.024,153.315
C02522=1083.980,42.170,439.200,174.456,20.022,153.315
C02523=1083.974,41.920,439.216,174.454,20.019,153.315
C02524=1083.968,41.671,439.231,174.453,20.017,153.314
C02525=1083.962,41.422,439.247,174.451,20.015,153.314
C02526=1083.957,41.172,439.263,174.449,20.013,153.314
C02527=1083.951,40.922,439.278,174.448,20.011,153.314
C02528=1083.946,40.674,439.294,174.446,20.009,153.314
C02529=1083.939,40.424,439.309,174.445,20.007,153.314
C02530=1083.933,40.175,439.325,174.444,20.005,153.314
C02531=1083.928,39.925,439.341,174.441,20.002,153.313
C02532=1083.923,39.675,439.356,174.440,20.000,153.313
C02533=1083.917,39.426,439.372,174.439,19.999,153.313
C02534=1083.910,39.176,439.387,174.437,19.996,153.313
C02535=1083.905,38.927,439.403,174.435,19.994,153.313
C02536=1083.899,38.678,439.419,174.433,19.992,153.313
C02537=1083.894,38.428,439.434,174.432,19.990,153.313
C02538=1083.888,38.179,439.449,174.431,19.988,153.312
C02539=1083.882,37.929,439.465,174.429,19.985,153.312
C02540=1083.876,37.679,439.481,174.427,19.983,153.312
C02541=1083.871,37.430,439.496,174.426,19.982,153.312
C02542=1083.864,37.181,439.512,174.424,19.979,153.312
C02543=1083.859,36.931,439.527,174.423,19.977,153.312
C02544=1083.853,36.682,439.542,174.421,19.975,153.311
C02545=1083.847,36.432,439.557,174.419,19.973,153.311
C02546=1083.841,36.183,439.574,174.418,19.971,153.311
C02547=1083.836,35.934,439.588,174.416,19.969,153.311
C02548=1083.830,35.684,439.604,174.414,19.967,153.311
C02549=1083.824,35.434,439.619,174.413,19.965,153.311
C02550=1083.818,35.186,439.634,174.412,19.963,153.311
C02551=1083.813,34.936,439.650,174.410,19.960,153.311
C02552=1083.806,34.686,439.665,174.408,19.958,153.310
C02553=1083.801,34.437,439.680,174.407,19.957,153.310
C02554=1083.795,34.187,439.696,174.405,19.954,153.310
C02555=1083.789,33.939,439.711,174.404,19.952,153.310
C02556=1083.784,33.689,439.727,174.402,19.950,153.310
C02557=1083.777,33.439,439.741,174.400,19.948,153.310
C02558=1083.772,33.190,439.757,174.399,19.946,153.309
C02559=1083.766,32.940,439.772,174.398,19.944,153.309
C02560=1083.760,32.691,439.788,174.395,19.942,153.309
C02561=1083.755,32.441,439.803,174.394,19.940,153.309
C02562=1083.749,32.192,439.818,174.393,19.938,153.309
C02563=1083.744,31.942,439.833,174.391,19.935,153.309
C02564=1083.737,31.693,439.848,174.390,19.933,153.309
C02565=1083.731,31.413,439.865,174.387,19.931,153.308
C02566=1083.725,31.135,439.882,174.386,19.929,153.308
C02567=1083.718,30.856,439.900,174.384,19.926,153.308
C02568=1083.712,30.578,439.916,174.382,19.924,153.308
C02569=1083.705,30.328,439.931,174.381,19.922,153.308
C02570=1083.700,30.079,439.947,174.379,19.920,153.308
C02571=1083.695,29.829,439.962,174.377,19.917,153.308
C02572=1083.689,29.580,439.977,174.376,19.915,153.307
C02573=1083.683,29.330,439.992,174.375,19.913,153.307
C02574=1083.677,29.081,440.007,174.373,19.911,153.307
C02575=1083.672,28.831,440.022,174.371,19.909,153.307
C02576=1083.665,28.581,440.037,174.370,19.907,153.307
C02577=1083.660,28.332,440.052,174.368,19.904,153.307
C02578=1083.654,28.082,440.067,174.367,19.903,153.307
C02579=1083.648,27.833,440.082,174.365,19.901,153.306
C02580=1083.643,27.583,440.098,174.363,19.898,153.306
C02581=1083.637,27.334,440.112,174.362,19.896,153.306
C02582=1083.631,27.084,440.128,174.361,19.894,153.306
C02583=1083.625,26.836,440.142,174.359,19.892,153.306
C02584=1083.619,26.586,440.157,174.357,19.890,153.306
C02585=1083.613,26.336,440.173,174.356,19.888,153.305
C02586=1083.608,26.087,440.187,174.355,19.886,153.305
C02587=1083.602,25.837,440.203,174.353,19.884,153.305
C02588=1083.596,25.588,440.217,174.351,19.882,153.305
C02589=1083.590,25.338,440.232,174.350,19.880,153.305
C02590=1083.585,25.089,440.248,174.348,19.877,153.305
C02591=1083.579,24.839,440.262,174.347,19.875,153.305
C02592=1083.573,24.590,440.276,174.345,19.873,153.304
C02593=1083.567,24.340,440.292,174.343,19.871,153.304
C02594=1083.561,24.091,440.306,174.342,19.869,153.304
C02595=1083.555,23.841,440.321,174.341,19.867,153.304
C02596=1083.550,23.592,440.337,174.338,19.865,153.304
C02597=1083.544,23.342,440.352,174.337,19.863,153.304
C02598=1083.538,23.093,440.366,174.336,19.861,153.303
C02599=1083.533,22.843,440.381,174.335,19.859,153.303
C02600=1083.527,22.594,440.396,174.333,19.856,153.303
C02601=1083.520,22.344,440.410,174.331,19.854,153.303
C02602=1083.515,22.095,440.426,174.330,19.852,153.303
C02603=1083.509,21.845,440.441,174.328,19.850,153.303
C02604=1083.503,21.596,440.454,174.327,19.848,153.303
C02605=1083.498,21.346,440.470,174.325,19.846,153.302
C02606=1083.492,21.097,440.485,174.323,19.844,153.302
C02607=1083.486,20.848,440.499,174.322,19.842,153.302
C02608=1083.480,20.598,440.514,174.321,19.840,153.302
C02609=1083.475,20.348,440.529,174.319,19.837,153.302
C02610=1083.469,20.099,440.544,174.317,19.835,153.302
C02611=1083.463,19.850,440.558,174.316,19.833,153.301
C02612=1083.457,19.600,440.573,174.315,19.831,153.301
C02613=1083.452,19.350,440.588,174.313,19.829,153.301
C02614=1083.445,19.100,440.602,174.311,19.827,153.301
C02615=1083.440,18.851,440.617,174.310,19.825,153.301
C02616=1083.433,18.602,440.632,174.308,19.823,153.301
C02617=1083.428,18.352,440.646,174.307,19.821,153.301
C02618=1083.423,18.103,440.661,174.305,19.819,153.300
C02619=1083.416,17.853,440.676,174.303,19.816,153.300
C02620=1083.411,17.604,440.690,174.302,19.814,153.300
C02621=1083.405,17.354,440.705,174.301,19.812,153.300
C02622=1083.399,17.105,440.719,174.299,19.811,153.300
C02623=1083.393,16.855,440.734,174.297,19.808,153.300
C02624=1083.388,16.606,440.749,174.296,19.806,153.300
C02625=1083.382,16.357,440.763,174.295,19.804,153.299
C02626=1083.376,16.106,440.778,174.293,19.802,153.299
C02627=1083.370,15.857,440.792,174.291,19.800,153.299
C02628=1083.364,15.607,440.806,174.290,19.798,153.299
C02629=1083.358,15.330,440.823,174.288,19.795,153.299
C02630=1083.351,15.053,440.839,174.287,19.793,153.299
C02631=1083.345,14.776,440.855,174.285,19.791,153.298
C02632=1083.339,14.498,440.871,174.283,19.789,153.298
C02633=1083.332,14.248,440.886,174.281,19.786,153.298
C02634=1083.327,13.999,440.900,174.280,19.784,153.298
C02635=1083.321,13.749,440.915,174.279,19.782,153.298
C02636=1083.315,13.500,440.929,174.278,19.780,153.298
C02637=1083.309,13.250,440.943,174.276,19.778,153.298
C02638=1083.303,13.001,440.958,174.274,19.776,153.297
C02639=1083.297,12.751,440.972,174.273,19.774,153.297
C02640=1083.291,12.502,440.987,174.271,19.772,153.297
C02641=1083.286,12.252,441.001,174.269,19.770,153.297
C02642=1083.279,12.003,441.016,174.268,19.768,153.297
C02643=1083.274,11.753,441.030,174.267,19.766,153.297
C02644=1083.268,11.504,441.044,174.265,19.764,153.297
C02645=1083.262,11.254,441.058,174.263,19.762,153.296
C02646=1083.256,11.005,441.073,174.262,19.760,153.296
C02647=1083.251,10.755,441.087,174.261,19.758,153.296
C02648=1083.244,10.506,441.102,174.259,19.755,153.296
C02649=1083.238,10.256,441.115,174.258,19.753,153.296
C02650=1083.232,10.006,441.129,174.256,19.751,153.296
C02651=1083.226,9.757,441.144,174.254,19.749,153.296
C02652=1083.221,9.508,441.158,174.253,19.747,153.295
C02653=1083.214,9.258,441.173,174.252,19.745,153.295
C02654=1083.209,9.008,441.186,174.250,19.743,153.295
C02655=1083.203,8.759,441.201,174.248,19.741,153.295
C02656=1083.197,8.509,441.215,174.247,19.739,153.295
C02657=1083.192,8.259,441.229,174.246,19.737,153.295
C02658=1083.186,8.011,441.244,174.244,19.735,153.295
C02659=1083.180,7.760,441.258,174.242,19.733,153.294
C02660=1083.174,7.511,441.272,174.241,19.731,153.294
C02661=1083.168,7.262,441.286,174.240,19.729,153.294
C02662=1083.162,7.012,441.300,174.238,19.726,153.294
C02663=1083.156,6.763,441.315,174.236,19.724,153.294
C02664=1083.150,6.513,441.328,174.235,19.722,153.294
C02665=1083.145,6.264,441.342,174.234,19.721,153.294
C02666=1083.138,6.014,441.357,174.231,19.718,153.293
C02667=1083.133,5.764,441.371,174.230,19.716,153.293
C02668=1083.128,5.515,441.385,174.229,19.714,153.293
C02669=1083.122,5.265,441.399,174.228,19.712,153.293
C02670=1083.115,5.016,441.413,174.226,19.710,153.293
C02671=1083.109,4.766,441.427,174.224,19.708,153.293
C02672=1083.104,4.517,441.441,174.223,19.705,153.292
C02673=1083.098,4.268,441.456,174.222,19.703,153.292
C02674=1083.092,4.018,441.470,174.220,19.702,153.292
C02675=1083.087,3.768,441.484,174.218,19.699,153.292
C02676=1083.081,3.518,441.498,174.217,19.697,153.292
C02677=1083.075,3.270,441.511,174.216,19.695,153.292
C02678=1083.069,3.019,441.526,174.214,19.693,153.292
C02679=1083.063,2.770,441.540,174.213,19.691,153.291
C02680=1083.058,2.520,441.553,174.211,19.689,153.291
C02681=1083.052,2.271,441.567,174.210,19.687,153.291
C02682=1083.046,2.021,441.582,174.208,19.684,153.291
C02683=1083.040,1.772,441.596,174.206,19.683,153.291
C02684=1083.034,1.522,441.609,174.205,19.681,153.291
C02685=1083.029,1.273,441.623,174.204,19.679,153.290
C02686=1083.023,1.023,441.637,174.202,19.676,153.290
C02687=1083.017,0.773,441.652,174.201,19.674,153.290
C02688=1083.011,0.524,441.666,174.199,19.672,153.290
C02689=1083.005,0.275,441.679,174.197,19.670,153.290
C02690=1083.000,0.025,441.693,174.196,19.668,153.290
C02691=1082.994,-0.225,441.707,174.195,19.666,153.290
C02692=1082.989,-0.474,441.721,174.194,19.664,153.289
C02693=1082.982,-0.750,441.736,174.192,19.661,153.289
C02694=1082.976,-1.025,441.751,174.190,19.659,153.289
C02695=1082.969,-1.301,441.767,174.188,19.657,153.289
C02696=1082.963,-1.575,441.782,174.187,19.655,153.289
C02697=1082.957,-1.825,441.796,174.186,19.653,153.289
C02698=1082.951,-2.075,441.810,174.184,19.650,153.288
C02699=1082.945,-2.325,441.824,174.182,19.648,153.288
C02700=1082.940,-2.574,441.838,174.181,19.646,153.288
C02701=1082.934,-2.824,441.851,174.180,19.645,153.288
C02702=1082.928,-3.073,441.865,174.178,19.642,153.288
C02703=1082.923,-3.323,441.879,174.176,19.640,153.288
C02704=1082.917,-3.572,441.892,174.175,19.638,153.288
C02705=1082.911,-3.822,441.907,174.174,19.636,153.287
C02706=1082.905,-4.072,441.920,174.172,19.634,153.287
C02707=1082.899,-4.321,441.934,174.170,19.632,153.287
C02708=1082.893,-4.571,441.948,174.169,19.630,153.287
C02709=1082.887,-4.820,441.961,174.168,19.628,153.287
C02710=1082.881,-5.070,441.975,174.166,19.626,153.287
C02711=1082.875,-5.320,441.988,174.165,19.624,153.287
C02712=1082.869,-5.569,442.002,174.163,19.622,153.286
C02713=1082.863,-5.818,442.016,174.162,19.620,153.286
C02714=1082.858,-6.068,442.029,174.161,19.618,153.286
C02715=1082.851,-6.317,442.043,174.158,19.616,153.286
C02716=1082.846,-6.567,442.057,174.157,19.613,153.286
C02717=1082.840,-6.817,442.071,174.156,19.612,153.286
C02718=1082.834,-7.066,442.084,174.155,19.610,153.286
C02719=1082.828,-7.316,442.098,174.152,19.607,153.285
C02720=1082.822,-7.565,442.111,174.151,19.605,153.285
C02721=1082.817,-7.815,442.124,174.150,19.603,153.285
C02722=1082.811,-8.065,442.138,174.148,19.602,153.285
C02723=1082.805,-8.314,442.151,174.146,19.599,153.285
C02724=1082.799,-8.563,442.165,174.145,19.597,153.285
C02725=1082.793,-8.814,442.179,174.144,19.595,153.285
C02726=1082.787,-9.063,442.192,174.143,19.593,153.284
C02727=1082.781,-9.313,442.206,174.141,19.591,153.284
C02728=1082.775,-9.562,442.219,174.139,19.589,153.284
C02729=1082.770,-9.812,442.232,174.138,19.587,153.284
C02730=1082.764,-10.061,442.246,174.137,19.585,153.284
C02731=1082.758,-10.311,442.260,174.135,19.583,153.284
C02732=1082.752,-10.560,442.273,174.133,19.581,153.284
C02733=1082.746,-10.810,442.287,174.132,19.579,153.284
C02734=1082.740,-11.059,442.300,174.131,19.577,153.283
C02735=1082.735,-11.309,442.313,174.129,19.575,153.283
C02736=1082.729,-11.558,442.326,174.128,19.573,153.283
C02737=1082.723,-11.808,442.340,174.126,19.571,153.283
C02738=1082.717,-12.058,442.354,174.125,19.569,153.283
C02739=1082.710,-12.307,442.367,174.123,19.567,153.283
C02740=1082.705,-12.557,442.380,174.122,19.565,153.283
C02741=1082.699,-12.807,442.394,174.120,19.563,153.282
C02742=1082.693,-13.056,442.407,174.119,19.561,153.282
C02743=1082.687,-13.306,442.421,174.117,19.559,153.282
C02744=1082.682,-13.556,442.434,174.116,19.557,153.282
C02745=1082.676,-13.805,442.447,174.115,19.555,153.282
C02746=1082.670,-14.055,442.461,174.113,19.553,153.282
C02747=1082.664,-14.304,442.474,174.112,19.551,153.282
C02748=1082.658,-14.554,442.487,174.110,19.549,153.281
C02749=1082.653,-14.803,442.501,174.109,19.547,153.281
C02750=1082.647,-15.053,442.514,174.108,19.545,153.281
C02751=1082.641,-15.303,442.527,174.106,19.542,153.281
C02752=1082.635,-15.552,442.540,174.104,19.540,153.281
C02753=1082.629,-15.801,442.554,174.103,19.539,153.281
C02754=1082.623,-16.051,442.566,174.102,19.537,153.281
C02755=1082.618,-16.301,442.580,174.100,19.535,153.280
C02756=1082.611,-16.550,442.593,174.098,19.533,153.280
C02757=1082.605,-16.824,442.607,174.097,19.531,153.280
C02758=1082.598,-17.097,442.622,174.095,19.528,153.280
C02759=1082.592,-17.372,442.636,174.094,19.526,153.280
C02760=1082.586,-17.645,442.651,174.092,19.524,153.280
C02761=1082.580,-17.895,442.664,174.090,19.522,153.280
C02762=1082.573,-18.144,442.677,174.089,19.520,153.280
C02763=1082.568,-18.394,442.691,174.087,19.518,153.279
C02764=1082.562,-18.644,442.703,174.086,19.516,153.279
C02765=1082.556,-18.893,442.717,174.085,19.514,153.279
C02766=1082.550,-19.143,442.729,174.083,19.512,153.279
C02767=1082.545,-19.392,442.743,174.081,19.510,153.279
C02768=1082.539,-19.642,442.755,174.080,19.508,153.279
C02769=1082.532,-19.892,442.769,174.079,19.506,153.279
C02770=1082.526,-20.141,442.781,174.078,19.505,153.279
C02771=1082.521,-20.391,442.795,174.075,19.502,153.278
C02772=1082.515,-20.640,442.808,174.074,19.500,153.278
C02773=1082.509,-20.890,442.821,174.073,19.499,153.278
C02774=1082.503,-21.139,442.834,174.072,19.497,153.278
C02775=1082.497,-21.389,442.847,174.070,19.495,153.278
C02776=1082.491,-21.639,442.861,174.069,19.493,153.278
C02777=1082.485,-21.889,442.873,174.067,19.491,153.278
C02778=1082.479,-22.138,442.887,174.066,19.489,153.278
C02779=1082.473,-22.388,442.899,174.064,19.487,153.277
C02780=1082.467,-22.637,442.912,174.063,19.485,153.277
C02781=1082.462,-22.887,442.925,174.062,19.483,153.277
C02782=1082.456,-23.137,442.938,174.060,19.480,153.277
C02783=1082.450,-23.386,442.951,174.058,19.478,153.277
C02784=1082.444,-23.636,442.963,174.057,19.477,153.277
C02785=1082.438,-23.885,442.977,174.056,19.475,153.277
C02786=1082.432,-24.135,442.989,174.054,19.473,153.276
C02787=1082.427,-24.384,443.003,174.052,19.471,153.276
C02788=1082.421,-24.634,443.016,174.051,19.469,153.276
C02789=1082.415,-24.884,443.028,174.050,19.467,153.276
C02790=1082.409,-25.133,443.042,174.048,19.465,153.276
C02791=1082.403,-25.383,443.054,174.047,19.463,153.276
C02792=1082.397,-25.632,443.067,174.046,19.461,153.276
C02793=1082.392,-25.882,443.080,174.044,19.459,153.276
C02794=1082.386,-26.132,443.093,174.042,19.457,153.276
C02795=1082.380,-26.381,443.106,174.041,19.455,153.275
C02796=1082.374,-26.631,443.119,174.040,19.453,153.275
C02797=1082.368,-26.881,443.131,174.038,19.452,153.275
C02798=1082.362,-27.130,443.144,174.036,19.449,153.275
C02799=1082.356,-27.380,443.157,174.035,19.447,153.275
C02800=1082.351,-27.629,443.169,174.033,19.446,153.275
C02801=1082.345,-27.879,443.182,174.032,19.444,153.275
C02802=1082.339,-28.129,443.195,174.031,19.442,153.274
C02803=1082.333,-28.378,443.207,174.029,19.440,153.274
C02804=1082.327,-28.628,443.221,174.027,19.438,153.274
C02805=1082.321,-28.878,443.233,174.026,19.436,153.274
C02806=1082.315,-29.127,443.246,174.025,19.434,153.274
C02807=1082.308,-29.377,443.259,174.023,19.432,153.274
C02808=1082.303,-29.627,443.272,174.022,19.431,153.274
C02809=1082.297,-29.876,443.284,174.021,19.428,153.274
C02810=1082.291,-30.126,443.296,174.018,19.426,153.274
C02811=1082.285,-30.375,443.310,174.017,19.424,153.274
C02812=1082.279,-30.625,443.322,174.016,19.422,153.273
C02813=1082.273,-30.875,443.335,174.015,19.421,153.273
C02814=1082.267,-31.124,443.347,174.013,19.419,153.273
C02815=1082.260,-31.374,443.360,174.012,19.417,153.273
C02816=1082.255,-31.623,443.372,174.010,19.415,153.273
C02817=1082.249,-31.873,443.385,174.009,19.413,153.273
C02818=1082.243,-32.122,443.397,174.007,19.411,153.273
C02819=1082.237,-32.372,443.410,174.006,19.409,153.273
C02820=1082.231,-32.622,443.423,174.004,19.408,153.273
C02821=1082.225,-32.895,443.437,174.002,19.405,153.272
C02822=1082.218,-33.167,443.450,174.001,19.403,153.272
C02823=1082.213,-33.441,443.464,174.000,19.401,153.272
C02824=1082.205,-33.714,443.478,173.998,19.399,153.272
C02825=1082.200,-33.963,443.490,173.996,19.397,153.272
C02826=1082.194,-34.213,443.503,173.995,19.395,153.272
C02827=1082.188,-34.463,443.515,173.994,19.394,153.272
C02828=1082.182,-34.712,443.528,173.992,19.392,153.272
C02829=1082.177,-34.962,443.540,173.991,19.390,153.272
C02830=1082.171,-35.212,443.552,173.989,19.388,153.271
C02831=1082.165,-35.461,443.565,173.987,19.386,153.271
C02832=1082.159,-35.711,443.578,173.986,19.384,153.271
C02833=1082.152,-35.960,443.590,173.985,19.382,153.271
C02834=1082.147,-36.209,443.602,173.984,19.381,153.271
C02835=1082.141,-36.459,443.615,173.982,19.378,153.271
C02836=1082.135,-36.709,443.628,173.981,19.377,153.271
C02837=1082.130,-36.958,443.640,173.979,19.374,153.271
C02838=1082.124,-37.208,443.652,173.978,19.372,153.270
C02839=1082.118,-37.458,443.665,173.976,19.371,153.270
C02840=1082.112,-37.708,443.677,173.975,19.369,153.270
C02841=1082.106,-37.957,443.689,173.973,19.367,153.270
C02842=1082.100,-38.207,443.702,173.972,19.365,153.270
C02843=1082.094,-38.457,443.714,173.971,19.364,153.270
C02844=1082.088,-38.707,443.727,173.969,19.361,153.270
C02845=1082.083,-38.956,443.739,173.967,19.360,153.270
C02846=1082.076,-39.205,443.751,173.966,19.358,153.270
C02847=1082.070,-39.455,443.763,173.964,19.356,153.270
C02848=1082.064,-39.705,443.776,173.963,19.354,153.269
C02849=1082.058,-39.954,443.788,173.962,19.353,153.269
C02850=1082.052,-40.204,443.800,173.961,19.351,153.269
C02851=1082.046,-40.454,443.813,173.958,19.349,153.269
C02852=1082.040,-40.703,443.825,173.957,19.347,153.269
C02853=1082.035,-40.952,443.837,173.956,19.345,153.269
C02854=1082.029,-41.202,443.849,173.954,19.343,153.269
C02855=1082.022,-41.452,443.861,173.953,19.342,153.269
C02856=1082.016,-41.702,443.874,173.952,19.340,153.269
C02857=1082.011,-41.951,443.886,173.950,19.338,153.269
C02858=1082.004,-42.201,443.898,173.949,19.336,153.268
C02859=1081.998,-42.451,443.910,173.947,19.334,153.269
C02860=1081.993,-42.700,443.922,173.945,19.333,153.268
C02861=1081.987,-42.950,443.934,173.944,19.331,153.268
C02862=1081.981,-43.200,443.947,173.943,19.329,153.268
C02863=1081.975,-43.450,443.959,173.941,19.327,153.268
C02864=1081.969,-43.698,443.971,173.940,19.325,153.268
C02865=1081.963,-43.948,443.983,173.939,19.323,153.268
C02866=1081.957,-44.198,443.996,173.937,19.322,153.268
C02867=1081.951,-44.448,444.007,173.935,19.319,153.268
C02868=1081.945,-44.698,444.019,173.934,19.318,153.268
C02869=1081.939,-44.947,444.031,173.932,19.316,153.268
C02870=1081.933,-45.196,444.043,173.931,19.314,153.267
C02871=1081.927,-45.446,444.056,173.929,19.313,153.267
C02872=1081.921,-45.696,444.068,173.928,19.311,153.267
C02873=1081.916,-45.946,444.079,173.927,19.309,153.267
C02874=1081.910,-46.195,444.092,173.926,19.307,153.267
C02875=1081.903,-46.445,444.104,173.923,19.305,153.267
C02876=1081.898,-46.694,444.116,173.922,19.304,153.267
C02877=1081.891,-46.944,444.128,173.921,19.302,153.267
C02878=1081.886,-47.194,444.139,173.919,19.300,153.267
C02879=1081.880,-47.443,444.152,173.918,19.298,153.267
C02880=1081.874,-47.693,444.164,173.916,19.297,153.267
C02881=1081.868,-47.942,444.176,173.915,19.295,153.266
C02882=1081.862,-48.192,444.187,173.914,19.293,153.266
C02883=1081.856,-48.442,444.200,173.912,19.292,153.266
C02884=1081.850,-48.691,444.212,173.910,19.289,153.266
C02885=1081.844,-48.964,444.225,173.909,19.288,153.266
C02886=1081.837,-49.239,444.238,173.908,19.286,153.266
C02887=1081.831,-49.512,444.251,173.906,19.284,153.266
C02888=1081.825,-49.785,444.264,173.904,19.282,153.266
C02889=1081.818,-50.035,444.276,173.903,19.280,153.266
C02890=1081.813,-50.284,444.288,173.901,19.278,153.266
C02891=1081.806,-50.534,444.300,173.900,19.276,153.266
C02892=1081.801,-50.784,444.312,173.898,19.275,153.266
C02893=1081.795,-51.033,444.323,173.897,19.273,153.265
C02894=1081.788,-51.283,444.335,173.896,19.271,153.265
C02895=1081.782,-51.533,444.347,173.894,19.270,153.265
C02896=1081.777,-51.782,444.358,173.892,19.268,153.265
C02897=1081.770,-52.032,444.370,173.891,19.266,153.265
C02898=1081.765,-52.281,444.383,173.889,19.264,153.265
C02899=1081.758,-52.531,444.394,173.888,19.263,153.265
C02900=1081.752,-52.781,444.406,173.886,19.261,153.265
C02901=1081.746,-53.030,444.418,173.885,19.259,153.265
C02902=1081.740,-53.280,444.429,173.884,19.258,153.265
C02903=1081.733,-53.530,444.441,173.882,19.256,153.265
C02904=1081.728,-53.780,444.453,173.881,19.255,153.265
C02905=1081.722,-54.029,444.465,173.880,19.253,153.265
C02906=1081.716,-54.278,444.476,173.878,19.251,153.265
C02907=1081.709,-54.528,444.487,173.877,19.250,153.265
C02908=1081.703,-54.778,444.500,173.874,19.248,153.265
C02909=1081.698,-55.028,444.511,173.873,19.246,153.264
C02910=1081.691,-55.277,444.523,173.872,19.244,153.264
C02911=1081.686,-55.527,444.534,173.870,19.243,153.264
C02912=1081.679,-55.777,444.546,173.869,19.241,153.264
C02913=1081.673,-56.027,444.557,173.867,19.239,153.264
C02914=1081.667,-56.276,444.569,173.866,19.238,153.264
C02915=1081.661,-56.526,444.581,173.865,19.236,153.264
C02916=1081.655,-56.775,444.592,173.863,19.235,153.264
C02917=1081.649,-57.025,444.604,173.862,19.233,153.264
C02918=1081.643,-57.274,444.615,173.860,19.231,153.264
C02919=1081.637,-57.525,444.627,173.859,19.229,153.264
C02920=1081.631,-57.774,444.639,173.858,19.228,153.264
C02921=1081.625,-58.024,444.650,173.855,19.226,153.264
C02922=1081.619,-58.273,444.663,173.854,19.224,153.264
C02923=1081.613,-58.523,444.673,173.853,19.222,153.264
C02924=1081.607,-58.773,444.685,173.851,19.221,153.264
C02925=1081.601,-59.022,444.696,173.850,19.219,153.264
C02926=1081.594,-59.272,444.708,173.848,19.218,153.264
C02927=1081.589,-59.521,444.720,173.847,19.216,153.264
C02928=1081.583,-59.771,444.732,173.845,19.214,153.263
C02929=1081.577,-60.020,444.743,173.844,19.213,153.263
C02930=1081.571,-60.271,444.754,173.843,19.211,153.263
C02931=1081.565,-60.520,444.766,173.841,19.210,153.263
C02932=1081.559,-60.770,444.777,173.840,19.208,153.263
C02933=1081.553,-61.019,444.789,173.838,19.207,153.263
C02934=1081.546,-61.269,444.800,173.837,19.205,153.263
C02935=1081.541,-61.519,444.811,173.836,19.203,153.263
C02936=1081.535,-61.768,444.823,173.833,19.201,153.263
C02937=1081.529,-62.018,444.834,173.832,19.200,153.263
C02938=1081.523,-62.268,444.846,173.830,19.198,153.263
C02939=1081.517,-62.517,444.857,173.829,19.197,153.263
C02940=1081.510,-62.767,444.868,173.828,19.195,153.263
C02941=1081.505,-63.017,444.880,173.826,19.193,153.263
C02942=1081.499,-63.267,444.892,173.825,19.192,153.263
C02943=1081.493,-63.516,444.903,173.823,19.190,153.263
C02944=1081.487,-63.766,444.914,173.822,19.189,153.263
C02945=1081.481,-64.015,444.926,173.820,19.187,153.263
C02946=1081.476,-64.265,444.937,173.819,19.186,153.263
C02947=1081.469,-64.515,444.948,173.818,19.184,153.262
C02948=1081.463,-64.764,444.960,173.816,19.182,153.262
C02949=1081.457,-65.039,444.972,173.815,19.181,153.262
C02950=1081.450,-65.314,444.985,173.812,19.179,153.262
C02951=1081.444,-65.589,444.997,173.811,19.177,153.262
C02952=1081.437,-65.863,445.009,173.810,19.175,153.262
C02953=1081.431,-66.113,445.021,173.808,19.173,153.262
C02954=1081.425,-66.363,445.031,173.807,19.172,153.262
C02955=1081.419,-66.612,445.044,173.805,19.170,153.262
C02956=1081.413,-66.862,445.055,173.804,19.169,153.262
C02957=1081.407,-67.111,445.066,173.802,19.167,153.262
C02958=1081.401,-67.362,445.077,173.801,19.166,153.262
C02959=1081.395,-67.611,445.088,173.800,19.164,153.262
C02960=1081.389,-67.860,445.100,173.797,19.162,153.262
C02961=1081.383,-68.110,445.111,173.796,19.160,153.262
C02962=1081.378,-68.360,445.122,173.795,19.159,153.262
C02963=1081.372,-68.610,445.133,173.793,19.157,153.262
C02964=1081.366,-68.860,445.144,173.792,19.156,153.262
C02965=1081.360,-69.108,445.156,173.790,19.154,153.262
C02966=1081.354,-69.359,445.167,173.789,19.153,153.262
C02967=1081.348,-69.608,445.178,173.787,19.151,153.262
C02968=1081.342,-69.858,445.189,173.786,19.150,153.262
C02969=1081.336,-70.108,445.200,173.784,19.148,153.262
C02970=1081.331,-70.358,445.212,173.783,19.147,153.262
C02971=1081.325,-70.607,445.223,173.781,19.145,153.262
C02972=1081.318,-70.857,445.235,173.780,19.144,153.261
C02973=1081.313,-71.106,445.245,173.779,19.142,153.261
C02974=1081.307,-71.356,445.256,173.777,19.140,153.261
C02975=1081.301,-71.606,445.267,173.776,19.139,153.261
C02976=1081.295,-71.855,445.278,173.774,19.137,153.261
C02977=1081.289,-72.105,445.289,173.773,19.136,153.261
C02978=1081.283,-72.355,445.300,173.772,19.134,153.261
C02979=1081.277,-72.605,445.311,173.770,19.133,153.261
C02980=1081.271,-72.854,445.322,173.769,19.131,153.261
C02981=1081.266,-73.104,445.334,173.767,19.130,153.261
C02982=1081.260,-73.354,445.345,173.766,19.128,153.261
C02983=1081.254,-73.604,445.356,173.764,19.126,153.261
C02984=1081.248,-73.853,445.367,173.763,19.125,153.261
C02985=1081.242,-74.103,445.378,173.761,19.123,153.261
C02986=1081.236,-74.353,445.389,173.760,19.122,153.261
C02987=1081.231,-74.602,445.400,173.758,19.120,153.261
C02988=1081.224,-74.852,445.410,173.757,19.119,153.261
C02989=1081.218,-75.102,445.421,173.755,19.117,153.261
C02990=1081.212,-75.350,445.433,173.754,19.116,153.261
C02991=1081.206,-75.601,445.443,173.752,19.115,153.261
C02992=1081.200,-75.851,445.454,173.751,19.113,153.261
C02993=1081.194,-76.100,445.465,173.749,19.112,153.261
C02994=1081.188,-76.350,445.476,173.748,19.110,153.261
C02995=1081.182,-76.600,445.487,173.747,19.109,153.261
C02996=1081.176,-76.849,445.498,173.745,19.107,153.261
C02997=1081.170,-77.099,445.508,173.744,19.106,153.261
C02998=1081.164,-77.349,445.520,173.742,19.104,153.261
C02999=1081.158,-77.598,445.531,173.741,19.103,153.261
C03000=1081.152,-77.848,445.541,173.739,19.102,153.261
C03001=1081.146,-78.098,445.553,173.738,19.100,153.261
C03002=1081.140,-78.347,445.564,173.736,19.099,153.261
C03003=1081.134,-78.597,445.574,173.735,19.097,153.261
C03004=1081.128,-78.846,445.585,173.733,19.096,153.261
C03005=1081.121,-79.096,445.596,173.732,19.094,153.261
C03006=1081.116,-79.346,445.607,173.730,19.093,153.261
C03007=1081.110,-79.595,445.618,173.729,19.092,153.261
C03008=1081.105,-79.845,445.628,173.727,19.090,153.261
C03009=1081.097,-80.095,445.638,173.726,19.089,153.261
C03010=1081.092,-80.345,445.649,173.724,19.087,153.261
C03011=1081.086,-80.594,445.660,173.723,19.086,153.261
C03012=1081.079,-80.844,445.671,173.721,19.085,153.261
C03013=1081.073,-81.121,445.683,173.720,19.083,153.261
C03014=1081.065,-81.398,445.695,173.718,19.082,153.261
C03015=1081.059,-81.675,445.706,173.716,19.080,153.261
C03016=1081.052,-81.952,445.718,173.714,19.078,153.261
C03017=1081.046,-82.201,445.729,173.713,19.077,153.261
C03018=1081.040,-82.451,445.739,173.711,19.076,153.261
C03019=1081.034,-82.700,445.750,173.710,19.074,153.261
C03020=1081.028,-82.951,445.761,173.708,19.073,153.261
C03021=1081.021,-83.200,445.771,173.707,19.072,153.261
C03022=1081.016,-83.450,445.782,173.705,19.070,153.261
C03023=1081.009,-83.700,445.793,173.704,19.069,153.261
C03024=1081.003,-83.949,445.803,173.702,19.068,153.261
C03025=1080.997,-84.199,445.814,173.701,19.067,153.261
C03026=1080.992,-84.449,445.824,173.700,19.065,153.261
C03027=1080.985,-84.698,445.835,173.698,19.064,153.261
C03028=1080.979,-84.948,445.846,173.697,19.063,153.261
C03029=1080.973,-85.198,445.856,173.695,19.061,153.261
C03030=1080.967,-85.447,445.866,173.694,19.060,153.261
C03031=1080.961,-85.697,445.878,173.692,19.059,153.261
C03032=1080.954,-85.947,445.888,173.691,19.057,153.261
C03033=1080.949,-86.197,445.898,173.689,19.056,153.261
C03034=1080.943,-86.446,445.909,173.688,19.055,153.261
C03035=1080.937,-86.695,445.919,173.686,19.053,153.261
C03036=1080.931,-86.946,445.930,173.684,19.052,153.261
C03037=1080.924,-87.195,445.940,173.683,19.050,153.261
C03038=1080.918,-87.445,445.951,173.682,19.049,153.261
C03039=1080.913,-87.695,445.961,173.680,19.048,153.261
C03040=1080.906,-87.944,445.971,173.678,19.046,153.261
C03041=1080.900,-88.194,445.983,173.677,19.045,153.261
C03042=1080.894,-88.444,445.992,173.675,19.044,153.261
C03043=1080.888,-88.694,446.003,173.674,19.042,153.261
C03044=1080.882,-88.943,446.014,173.672,19.041,153.261
C03045=1080.876,-89.193,446.024,173.671,19.040,153.261
C03046=1080.870,-89.442,446.034,173.670,19.039,153.261
C03047=1080.863,-89.692,446.045,173.668,19.038,153.261
C03048=1080.858,-89.942,446.055,173.667,19.036,153.261
C03049=1080.851,-90.192,446.066,173.665,19.035,153.261
C03050=1080.846,-90.442,446.076,173.664,19.034,153.261
C03051=1080.840,-90.691,446.086,173.662,19.032,153.261
C03052=1080.834,-90.940,446.097,173.661,19.031,153.261
C03053=1080.828,-91.191,446.107,173.659,19.030,153.261
C03054=1080.821,-91.440,446.118,173.658,19.028,153.261
C03055=1080.816,-91.690,446.128,173.656,19.027,153.261
C03056=1080.809,-91.940,446.138,173.654,19.026,153.261
C03057=1080.804,-92.190,446.148,173.653,19.025,153.262
C03058=1080.798,-92.439,446.159,173.651,19.023,153.262
C03059=1080.792,-92.688,446.169,173.650,19.022,153.261
C03060=1080.786,-92.938,446.179,173.648,19.021,153.262
C03061=1080.779,-93.188,446.190,173.647,19.019,153.262
C03062=1080.773,-93.438,446.200,173.646,19.019,153.262
C03063=1080.767,-93.688,446.211,173.644,19.017,153.262
C03064=1080.762,-93.938,446.221,173.643,19.016,153.262
C03065=1080.755,-94.187,446.231,173.641,19.015,153.262
C03066=1080.750,-94.437,446.241,173.640,19.014,153.262
C03067=1080.744,-94.686,446.252,173.638,19.012,153.262
C03068=1080.738,-94.936,446.262,173.637,19.011,153.262
C03069=1080.732,-95.186,446.272,173.635,19.010,153.262
C03070=1080.726,-95.436,446.282,173.634,19.008,153.262
C03071=1080.720,-95.685,446.292,173.632,19.007,153.262
C03072=1080.714,-95.935,446.303,173.630,19.006,153.262
C03073=1080.708,-96.185,446.312,173.629,19.005,153.262
C03074=1080.702,-96.435,446.323,173.628,19.004,153.262
C03075=1080.696,-96.685,446.333,173.626,19.003,153.262
C03076=1080.690,-96.934,446.344,173.625,19.001,153.262
C03077=1080.684,-97.213,446.355,173.623,19.000,153.262
C03078=1080.677,-97.492,446.366,173.621,18.998,153.262
C03079=1080.670,-97.771,446.377,173.619,18.997,153.262
C03080=1080.663,-98.050,446.389,173.618,18.996,153.262
C03081=1080.657,-98.300,446.399,173.616,18.995,153.262
C03082=1080.651,-98.550,446.409,173.614,18.994,153.263
C03083=1080.645,-98.799,446.419,173.613,18.992,153.262
C03084=1080.638,-99.050,446.429,173.612,18.992,153.263
C03085=1080.632,-99.299,446.439,173.611,18.990,153.263
C03086=1080.626,-99.549,446.449,173.609,18.989,153.263
C03087=1080.620,-99.798,446.459,173.607,18.988,153.263
C03088=1080.614,-100.048,446.469,173.606,18.987,153.263
C03089=1080.608,-100.298,446.479,173.604,18.986,153.263
C03090=1080.601,-100.547,446.489,173.602,18.985,153.263
C03091=1080.596,-100.798,446.499,173.601,18.983,153.263
C03092=1080.590,-101.047,446.509,173.599,18.982,153.263
C03093=1080.583,-101.297,446.519,173.598,18.982,153.263
C03094=1080.577,-101.546,446.529,173.597,18.980,153.263
C03095=1080.572,-101.796,446.539,173.595,18.979,153.263
C03096=1080.565,-102.046,446.549,173.594,18.978,153.263
C03097=1080.559,-102.295,446.559,173.592,18.977,153.263
C03098=1080.554,-102.546,446.569,173.590,18.976,153.263
C03099=1080.548,-102.795,446.579,173.589,18.975,153.264
C03100=1080.541,-103.044,446.589,173.587,18.973,153.263
C03101=1080.535,-103.294,446.598,173.586,18.972,153.264
C03102=1080.529,-103.544,446.609,173.585,18.972,153.264
C03103=1080.523,-103.794,446.619,173.583,18.970,153.264
C03104=1080.517,-104.043,446.628,173.582,18.969,153.264
C03105=1080.511,-104.293,446.638,173.580,18.968,153.264
C03106=1080.505,-104.543,446.648,173.578,18.967,153.264
C03107=1080.499,-104.792,446.658,173.577,18.966,153.264
C03108=1080.493,-105.042,446.668,173.575,18.965,153.264
C03109=1080.486,-105.292,446.678,173.574,18.964,153.264
C03110=1080.481,-105.542,446.688,173.573,18.963,153.264
C03111=1080.475,-105.792,446.697,173.571,18.962,153.264
C03112=1080.468,-106.041,446.708,173.569,18.961,153.264
C03113=1080.462,-106.291,446.717,173.568,18.960,153.264
C03114=1080.456,-106.541,446.727,173.566,18.958,153.264
C03115=1080.450,-106.791,446.737,173.564,18.957,153.265
C03116=1080.444,-107.041,446.747,173.563,18.956,153.265
C03117=1080.438,-107.290,446.757,173.562,18.956,153.265
C03118=1080.432,-107.540,446.766,173.560,18.955,153.265
C03119=1080.426,-107.789,446.776,173.559,18.953,153.265
C03120=1080.419,-108.039,446.785,173.557,18.952,153.265
C03121=1080.413,-108.289,446.795,173.555,18.951,153.265
C03122=1080.408,-108.539,446.805,173.554,18.950,153.265
C03123=1080.402,-108.789,446.815,173.552,18.949,153.265
C03124=1080.395,-109.038,446.825,173.551,18.949,153.265
C03125=1080.389,-109.288,446.835,173.549,18.948,153.265
C03126=1080.383,-109.538,446.844,173.548,18.946,153.265
C03127=1080.377,-109.787,446.854,173.546,18.945,153.266
C03128=1080.370,-110.037,446.863,173.545,18.944,153.266
C03129=1080.364,-110.287,446.873,173.543,18.944,153.266
C03130=1080.358,-110.537,446.882,173.542,18.943,153.266
C03131=1080.352,-110.787,446.892,173.540,18.942,153.266
C03132=1080.346,-111.036,446.902,173.539,18.941,153.266
C03133=1080.340,-111.286,446.911,173.537,18.940,153.266
C03134=1080.334,-111.536,446.922,173.535,18.939,153.266
C03135=1080.328,-111.786,446.932,173.534,18.938,153.266
C03136=1080.321,-112.035,446.941,173.533,18.937,153.266
C03137=1080.315,-112.285,446.951,173.531,18.936,153.266
C03138=1080.309,-112.535,446.960,173.530,18.935,153.267
C03139=1080.304,-112.784,446.970,173.528,18.934,153.267
C03140=1080.297,-113.034,446.979,173.526,18.933,153.267
C03141=1080.290,-113.310,446.989,173.524,18.932,153.267
C03142=1080.284,-113.586,447.000,173.523,18.931,153.267
C03143=1080.276,-113.863,447.011,173.521,18.930,153.267
C03144=1080.270,-114.138,447.022,173.519,18.929,153.267
C03145=1080.264,-114.388,447.031,173.518,18.928,153.267
C03146=1080.258,-114.638,447.041,173.516,18.927,153.268
C03147=1080.252,-114.888,447.050,173.515,18.927,153.268
C03148=1080.246,-115.138,447.059,173.513,18.926,153.268
C03149=1080.240,-115.387,447.069,173.512,18.925,153.268
C03150=1080.234,-115.637,447.078,173.510,18.924,153.268
C03151=1080.228,-115.887,447.088,173.508,18.923,153.268
C03152=1080.222,-116.136,447.097,173.507,18.922,153.268
C03153=1080.216,-116.386,447.107,173.506,18.921,153.268
C03154=1080.209,-116.636,447.116,173.504,18.920,153.268
C03155=1080.202,-116.886,447.125,173.502,18.919,153.268
C03156=1080.196,-117.135,447.135,173.501,18.918,153.269
C03157=1080.190,-117.385,447.145,173.499,18.917,153.269
C03158=1080.185,-117.634,447.154,173.498,18.917,153.269
C03159=1080.178,-117.884,447.163,173.496,18.916,153.269
C03160=1080.172,-118.134,447.173,173.495,18.915,153.269
C03161=1080.166,-118.384,447.182,173.493,18.914,153.269
C03162=1080.160,-118.633,447.192,173.491,18.913,153.269
C03163=1080.154,-118.884,447.201,173.490,18.912,153.269
C03164=1080.148,-119.134,447.210,173.489,18.911,153.269
C03165=1080.142,-119.383,447.220,173.487,18.910,153.270
C03166=1080.135,-119.632,447.229,173.485,18.910,153.270
C03167=1080.129,-119.882,447.238,173.483,18.909,153.270
C03168=1080.123,-120.132,447.248,173.483,18.909,153.270
C03169=1080.117,-120.382,447.257,173.481,18.908,153.270
C03170=1080.111,-120.632,447.266,173.479,18.907,153.270
C03171=1080.105,-120.882,447.276,173.477,18.906,153.270
C03172=1080.099,-121.132,447.285,173.476,18.905,153.270
C03173=1080.092,-121.380,447.294,173.475,18.904,153.271
C03174=1080.086,-121.630,447.303,173.473,18.904,153.271
C03175=1080.080,-121.880,447.313,173.471,18.903,153.271
C03176=1080.074,-122.130,447.322,173.470,18.902,153.271
C03177=1080.068,-122.380,447.331,173.469,18.901,153.271
C03178=1080.062,-122.630,447.341,173.467,18.900,153.271
C03179=1080.056,-122.879,447.350,173.465,18.899,153.271
C03180=1080.050,-123.129,447.358,173.463,18.899,153.272
C03181=1080.043,-123.379,447.368,173.462,18.898,153.272
C03182=1080.037,-123.629,447.378,173.461,18.897,153.272
C03183=1080.031,-123.879,447.387,173.459,18.896,153.272
C03184=1080.025,-124.128,447.396,173.457,18.895,153.272
C03185=1080.019,-124.378,447.405,173.456,18.895,153.272
C03186=1080.013,-124.628,447.414,173.455,18.894,153.272
C03187=1080.007,-124.877,447.424,173.453,18.893,153.272
C03188=1080.000,-125.127,447.433,173.451,18.892,153.273
C03189=1079.994,-125.377,447.442,173.449,18.892,153.273
C03190=1079.988,-125.626,447.451,173.448,18.891,153.273
C03191=1079.982,-125.876,447.460,173.447,18.890,153.273
C03192=1079.976,-126.127,447.469,173.445,18.889,153.273
C03193=1079.969,-126.376,447.478,173.443,18.889,153.273
C03194=1079.963,-126.626,447.488,173.441,18.888,153.274
C03195=1079.958,-126.876,447.496,173.441,18.888,153.274
C03196=1079.951,-127.125,447.505,173.439,18.887,153.274
C03197=1079.945,-127.375,447.515,173.437,18.886,153.274
C03198=1079.939,-127.625,447.524,173.435,18.885,153.274
C03199=1079.933,-127.875,447.533,173.434,18.885,153.274
C03200=1079.927,-128.125,447.542,173.433,18.884,153.274
C03201=1079.925,-128.380,447.553,173.431,18.882,153.274
C03202=1079.926,-128.635,447.565,173.431,18.879,153.274
C03203=1079.930,-128.888,447.578,173.430,18.875,153.273
C03204=1079.938,-129.140,447.592,173.430,18.870,153.272
C03205=1079.540,-129.162,447.448,173.386,18.992,153.303
C03206=1079.532,-128.910,447.435,173.386,18.997,153.304
C03207=1079.528,-128.657,447.421,173.386,19.001,153.304
C03208=1079.527,-128.402,447.410,173.387,19.004,153.305
C03209=1079.528,-128.147,447.399,173.388,19.006,153.305
C03210=1079.533,-127.897,447.389,173.390,19.007,153.305
C03211=1079.540,-127.647,447.381,173.391,19.008,153.305
C03212=1079.546,-127.397,447.371,173.393,19.008,153.305
C03213=1079.552,-127.147,447.362,173.394,19.009,153.304
C03214=1079.558,-126.898,447.353,173.396,19.010,153.304
C03215=1079.564,-126.648,447.344,173.398,19.010,153.304
C03216=1079.570,-126.398,447.335,173.399,19.011,153.304
C03217=1079.577,-126.148,447.326,173.400,19.012,153.304
C03218=1079.583,-125.898,447.317,173.402,19.013,153.304
C03219=1079.589,-125.649,447.308,173.404,19.013,153.303
C03220=1079.595,-125.399,447.299,173.406,19.014,153.303
C03221=1079.601,-125.149,447.289,173.407,19.015,153.303
C03222=1079.608,-124.900,447.280,173.408,19.016,153.303
C03223=1079.614,-124.649,447.271,173.410,19.016,153.303
C03224=1079.620,-124.399,447.262,173.412,19.017,153.303
C03225=1079.626,-124.150,447.253,173.413,19.018,153.303
C03226=1079.632,-123.901,447.244,173.415,19.019,153.303
C03227=1079.638,-123.650,447.235,173.416,19.020,153.302
C03228=1079.644,-123.401,447.225,173.418,19.021,153.302
C03229=1079.651,-123.151,447.216,173.420,19.021,153.302
C03230=1079.656,-122.902,447.206,173.421,19.022,153.302
C03231=1079.662,-122.652,447.197,173.422,19.023,153.302
C03232=1079.669,-122.402,447.189,173.424,19.023,153.302
C03233=1079.675,-122.152,447.179,173.426,19.024,153.302
C03234=1079.681,-121.902,447.169,173.427,19.025,153.302
C03235=1079.688,-121.652,447.160,173.428,19.026,153.302
C03236=1079.693,-121.403,447.151,173.430,19.026,153.301
C03237=1079.699,-121.153,447.142,173.432,19.027,153.301
C03238=1079.705,-120.903,447.132,173.434,19.028,153.301
C03239=1079.712,-120.654,447.123,173.435,19.029,153.301
C03240=1079.718,-120.404,447.114,173.436,19.030,153.301
C03241=1079.724,-120.154,447.104,173.438,19.031,153.301
C03242=1079.730,-119.905,447.095,173.440,19.032,153.301
C03243=1079.736,-119.655,447.086,173.441,19.033,153.300
C03244=1079.742,-119.405,447.077,173.442,19.033,153.300
C03245=1079.748,-119.155,447.067,173.444,19.034,153.300
C03246=1079.754,-118.905,447.057,173.446,19.035,153.300
C03247=1079.761,-118.656,447.048,173.448,19.036,153.300
C03248=1079.767,-118.406,447.039,173.449,19.037,153.300
C03249=1079.774,-118.156,447.029,173.451,19.038,153.300
C03250=1079.779,-117.907,447.020,173.452,19.038,153.300
C03251=1079.785,-117.657,447.011,173.454,19.039,153.299
C03252=1079.791,-117.407,447.002,173.455,19.040,153.299
C03253=1079.797,-117.157,446.992,173.457,19.041,153.299
C03254=1079.804,-116.907,446.983,173.459,19.042,153.299
C03255=1079.810,-116.657,446.973,173.460,19.042,153.299
C03256=1079.816,-116.408,446.963,173.461,19.043,153.299
C03257=1079.822,-116.158,446.954,173.463,19.044,153.299
C03258=1079.828,-115.908,446.944,173.465,19.045,153.299
C03259=1079.834,-115.659,446.935,173.466,19.046,153.299
C03260=1079.840,-115.409,446.926,173.468,19.047,153.298
C03261=1079.846,-115.159,446.916,173.469,19.048,153.298
C03262=1079.852,-114.910,446.906,173.471,19.049,153.298
C03263=1079.858,-114.660,446.897,173.472,19.050,153.298
C03264=1079.865,-114.410,446.888,173.474,19.051,153.298
C03265=1079.871,-114.160,446.878,173.476,19.052,153.298
C03266=1079.878,-113.884,446.868,173.477,19.053,153.298
C03267=1079.884,-113.608,446.856,173.479,19.054,153.298
C03268=1079.891,-113.332,446.846,173.481,19.055,153.298
C03269=1079.898,-113.055,446.836,173.482,19.056,153.298
C03270=1079.904,-112.805,446.826,173.484,19.057,153.297
C03271=1079.910,-112.556,446.817,173.485,19.058,153.297
C03272=1079.916,-112.306,446.807,173.486,19.059,153.297
C03273=1079.922,-112.056,446.797,173.488,19.060,153.297
C03274=1079.929,-111.806,446.788,173.490,19.061,153.297
C03275=1079.935,-111.557,446.778,173.492,19.062,153.297
C03276=1079.941,-111.308,446.768,173.493,19.063,153.297
C03277=1079.947,-111.058,446.759,173.494,19.064,153.297
C03278=1079.953,-110.808,446.749,173.496,19.065,153.297
C03279=1079.959,-110.558,446.740,173.497,19.066,153.297
C03280=1079.965,-110.309,446.730,173.499,19.067,153.297
C03281=1079.971,-110.059,446.721,173.501,19.068,153.296
C03282=1079.977,-109.809,446.710,173.502,19.069,153.296
C03283=1079.983,-109.559,446.701,173.504,19.070,153.296
C03284=1079.989,-109.309,446.691,173.505,19.071,153.296
C03285=1079.995,-109.059,446.682,173.506,19.072,153.296
C03286=1080.002,-108.810,446.671,173.508,19.072,153.296
C03287=1080.008,-108.560,446.662,173.510,19.073,153.296
C03288=1080.014,-108.311,446.652,173.512,19.074,153.296
C03289=1080.020,-108.061,446.643,173.513,19.076,153.296
C03290=1080.027,-107.811,446.633,173.515,19.077,153.296
C03291=1080.033,-107.561,446.624,173.516,19.077,153.296
C03292=1080.039,-107.312,446.613,173.517,19.078,153.296
C03293=1080.045,-107.062,446.603,173.519,19.079,153.295
C03294=1080.051,-106.812,446.594,173.520,19.081,153.295
C03295=1080.057,-106.562,446.584,173.522,19.082,153.295
C03296=1080.063,-106.313,446.574,173.524,19.083,153.295
C03297=1080.069,-106.062,446.564,173.525,19.084,153.295
C03298=1080.075,-105.813,446.554,173.526,19.085,153.295
C03299=1080.081,-105.563,446.544,173.528,19.086,153.295
C03300=1080.087,-105.314,446.535,173.530,19.087,153.295
C03301=1080.094,-105.064,446.525,173.531,19.088,153.295
C03302=1080.099,-104.814,446.514,173.533,19.089,153.295
C03303=1080.106,-104.565,446.505,173.534,19.090,153.295
C03304=1080.112,-104.315,446.495,173.536,19.092,153.295
C03305=1080.118,-104.065,446.486,173.538,19.093,153.295
C03306=1080.124,-103.815,446.475,173.538,19.093,153.295
C03307=1080.130,-103.566,446.465,173.540,19.094,153.294
C03308=1080.136,-103.316,446.456,173.542,19.096,153.295
C03309=1080.142,-103.066,446.446,173.543,19.097,153.294
C03310=1080.148,-102.817,446.435,173.545,19.098,153.294
C03311=1080.154,-102.567,446.426,173.546,19.099,153.294
C03312=1080.160,-102.317,446.416,173.548,19.100,153.294
C03313=1080.166,-102.068,446.405,173.550,19.102,153.294
C03314=1080.172,-101.818,446.396,173.551,19.103,153.294
C03315=1080.178,-101.568,446.386,173.552,19.103,153.294
C03316=1080.184,-101.318,446.377,173.554,19.105,153.294
C03317=1080.190,-101.069,446.366,173.555,19.106,153.294
C03318=1080.196,-100.819,446.356,173.557,19.107,153.294
C03319=1080.203,-100.569,446.346,173.558,19.108,153.294
C03320=1080.209,-100.319,446.335,173.560,19.109,153.294
C03321=1080.215,-100.069,446.326,173.562,19.111,153.294
C03322=1080.222,-99.820,446.315,173.563,19.112,153.294
C03323=1080.228,-99.570,446.306,173.565,19.113,153.294
C03324=1080.233,-99.320,446.296,173.566,19.114,153.294
C03325=1080.240,-99.071,446.285,173.567,19.115,153.294
C03326=1080.246,-98.821,446.276,173.569,19.116,153.294
C03327=1080.251,-98.571,446.266,173.570,19.117,153.293
C03328=1080.258,-98.322,446.255,173.572,19.118,153.293
C03329=1080.264,-98.072,446.246,173.574,19.120,153.293
C03330=1080.271,-97.793,446.234,173.575,19.121,153.293
C03331=1080.277,-97.513,446.223,173.577,19.122,153.293
C03332=1080.284,-97.234,446.212,173.578,19.123,153.293
C03333=1080.291,-96.955,446.200,173.581,19.125,153.293
C03334=1080.296,-96.705,446.190,173.582,19.126,153.293
C03335=1080.303,-96.455,446.180,173.583,19.127,153.293
C03336=1080.308,-96.205,446.170,173.585,19.129,153.293
C03337=1080.315,-95.956,446.159,173.586,19.130,153.293
C03338=1080.320,-95.706,446.149,173.588,19.131,153.293
C03339=1080.327,-95.457,446.139,173.589,19.132,153.293
C03340=1080.333,-95.206,446.128,173.591,19.134,153.293
C03341=1080.339,-94.957,446.118,173.593,19.135,153.293
C03342=1080.344,-94.707,446.108,173.594,19.136,153.293
C03343=1080.351,-94.458,446.098,173.596,19.137,153.293
C03344=1080.356,-94.208,446.087,173.597,19.139,153.293
C03345=1080.363,-93.958,446.077,173.599,19.140,153.293
C03346=1080.368,-93.708,446.067,173.600,19.141,153.293
C03347=1080.375,-93.459,446.057,173.601,19.142,153.293
C03348=1080.380,-93.209,446.046,173.603,19.143,153.293
C03349=1080.387,-92.960,446.036,173.604,19.145,153.293
C03350=1080.393,-92.709,446.026,173.606,19.146,153.293
C03351=1080.399,-92.460,446.015,173.607,19.147,153.293
C03352=1080.405,-92.210,446.005,173.609,19.149,153.293
C03353=1080.411,-91.960,445.995,173.610,19.150,153.292
C03354=1080.417,-91.711,445.984,173.612,19.151,153.292
C03355=1080.422,-91.461,445.974,173.613,19.153,153.293
C03356=1080.429,-91.212,445.964,173.615,19.154,153.292
C03357=1080.434,-90.962,445.953,173.617,19.155,153.292
C03358=1080.441,-90.712,445.943,173.618,19.156,153.292
C03359=1080.447,-90.462,445.933,173.620,19.158,153.292
C03360=1080.453,-90.212,445.922,173.621,19.159,153.292
C03361=1080.459,-89.963,445.911,173.623,19.160,153.292
C03362=1080.464,-89.713,445.901,173.624,19.162,153.292
C03363=1080.471,-89.464,445.891,173.625,19.163,153.292
C03364=1080.477,-89.213,445.880,173.627,19.164,153.292
C03365=1080.483,-88.964,445.870,173.628,19.165,153.292
C03366=1080.489,-88.714,445.859,173.630,19.167,153.292
C03367=1080.495,-88.464,445.850,173.631,19.168,153.292
C03368=1080.501,-88.215,445.839,173.633,19.169,153.292
C03369=1080.507,-87.965,445.828,173.634,19.171,153.292
C03370=1080.514,-87.715,445.818,173.636,19.172,153.292
C03371=1080.519,-87.465,445.807,173.637,19.173,153.292
C03372=1080.526,-87.216,445.797,173.639,19.175,153.292
C03373=1080.531,-86.967,445.786,173.640,19.176,153.292
C03374=1080.537,-86.717,445.776,173.642,19.177,153.292
C03375=1080.544,-86.467,445.765,173.643,19.179,153.292
C03376=1080.550,-86.217,445.754,173.645,19.180,153.292
C03377=1080.556,-85.967,445.745,173.647,19.181,153.292
C03378=1080.562,-85.718,445.734,173.648,19.183,153.292
C03379=1080.568,-85.468,445.723,173.649,19.184,153.292
C03380=1080.574,-85.219,445.712,173.651,19.185,153.292
C03381=1080.580,-84.968,445.702,173.653,19.187,153.292
C03382=1080.586,-84.719,445.691,173.654,19.188,153.292
C03383=1080.593,-84.469,445.681,173.656,19.189,153.292
C03384=1080.598,-84.220,445.670,173.657,19.191,153.292
C03385=1080.605,-83.970,445.660,173.659,19.192,153.292
C03386=1080.610,-83.720,445.649,173.660,19.194,153.292
C03387=1080.617,-83.470,445.638,173.661,19.194,153.292
C03388=1080.623,-83.221,445.628,173.663,19.196,153.292
C03389=1080.629,-82.971,445.617,173.664,19.197,153.292
C03390=1080.634,-82.721,445.607,173.665,19.199,153.292
C03391=1080.641,-82.471,445.596,173.667,19.200,153.292
C03392=1080.647,-82.222,445.585,173.669,19.201,153.292
C03393=1080.653,-81.973,445.574,173.670,19.203,153.292
C03394=1080.660,-81.696,445.563,173.672,19.205,153.292
C03395=1080.666,-81.418,445.551,173.674,19.206,153.292
C03396=1080.674,-81.141,445.539,173.675,19.208,153.292
C03397=1080.680,-80.864,445.527,173.677,19.209,153.292
C03398=1080.687,-80.615,445.516,173.678,19.210,153.292
C03399=1080.693,-80.365,445.506,173.680,19.212,153.292
C03400=1080.698,-80.115,445.495,173.681,19.213,153.292
C03401=1080.705,-79.865,445.485,173.683,19.215,153.292
C03402=1080.711,-79.616,445.474,173.685,19.216,153.292
C03403=1080.717,-79.366,445.463,173.686,19.217,153.292
C03404=1080.723,-79.116,445.452,173.687,19.219,153.292
C03405=1080.729,-78.867,445.441,173.689,19.220,153.292
C03406=1080.735,-78.617,445.431,173.690,19.222,153.292
C03407=1080.741,-78.368,445.420,173.692,19.223,153.292
C03408=1080.747,-78.118,445.409,173.693,19.225,153.292
C03409=1080.753,-77.868,445.398,173.695,19.226,153.292
C03410=1080.759,-77.619,445.387,173.696,19.228,153.292
C03411=1080.765,-77.368,445.376,173.698,19.229,153.292
C03412=1080.771,-77.119,445.365,173.699,19.230,153.292
C03413=1080.777,-76.869,445.355,173.701,19.232,153.292
C03414=1080.783,-76.620,445.344,173.702,19.233,153.292
C03415=1080.789,-76.370,445.333,173.704,19.235,153.292
C03416=1080.795,-76.120,445.322,173.705,19.236,153.292
C03417=1080.801,-75.871,445.311,173.707,19.238,153.292
C03418=1080.807,-75.620,445.300,173.708,19.239,153.292
C03419=1080.813,-75.371,445.289,173.710,19.241,153.292
C03420=1080.818,-75.122,445.278,173.711,19.242,153.292
C03421=1080.825,-74.871,445.267,173.713,19.244,153.292
C03422=1080.831,-74.622,445.257,173.714,19.245,153.292
C03423=1080.837,-74.373,445.246,173.715,19.247,153.292
C03424=1080.843,-74.122,445.235,173.717,19.248,153.292
C03425=1080.849,-73.873,445.224,173.718,19.250,153.292
C03426=1080.855,-73.623,445.213,173.720,19.251,153.292
C03427=1080.861,-73.373,445.202,173.721,19.253,153.292
C03428=1080.867,-73.124,445.190,173.723,19.254,153.292
C03429=1080.872,-72.875,445.178,173.724,19.256,153.293
C03430=1080.879,-72.624,445.167,173.726,19.257,153.293
C03431=1080.884,-72.375,445.156,173.727,19.259,153.293
C03432=1080.890,-72.125,445.145,173.729,19.260,153.293
C03433=1080.896,-71.876,445.135,173.730,19.262,153.293
C03434=1080.902,-71.626,445.123,173.732,19.263,153.293
C03435=1080.908,-71.376,445.112,173.733,19.265,153.293
C03436=1080.914,-71.127,445.102,173.734,19.267,153.293
C03437=1080.920,-70.877,445.090,173.736,19.268,153.293
C03438=1080.926,-70.627,445.079,173.737,19.270,153.293
C03439=1080.932,-70.378,445.068,173.739,19.271,153.293
C03440=1080.937,-70.128,445.056,173.740,19.273,153.293
C03441=1080.943,-69.878,445.045,173.742,19.274,153.293
C03442=1080.949,-69.629,445.034,173.743,19.276,153.293
C03443=1080.955,-69.379,445.023,173.745,19.278,153.293
C03444=1080.961,-69.129,445.012,173.747,19.280,153.293
C03445=1080.967,-68.880,445.001,173.748,19.282,153.293
C03446=1080.973,-68.630,444.989,173.749,19.283,153.293
C03447=1080.979,-68.381,444.978,173.751,19.285,153.293
C03448=1080.985,-68.130,444.967,173.752,19.286,153.293
C03449=1080.990,-67.881,444.956,173.754,19.288,153.293
C03450=1080.996,-67.631,444.945,173.755,19.289,153.293
C03451=1081.003,-67.381,444.933,173.757,19.291,153.293
C03452=1081.008,-67.132,444.922,173.758,19.292,153.293
C03453=1081.015,-66.882,444.911,173.759,19.294,153.294
C03454=1081.021,-66.632,444.900,173.761,19.296,153.294
C03455=1081.026,-66.383,444.888,173.762,19.297,153.294
C03456=1081.032,-66.133,444.876,173.764,19.299,153.294
C03457=1081.038,-65.883,444.866,173.765,19.300,153.294
C03458=1081.045,-65.609,444.853,173.767,19.302,153.294
C03459=1081.051,-65.334,444.841,173.769,19.304,153.294
C03460=1081.058,-65.060,444.828,173.770,19.306,153.294
C03461=1081.065,-64.784,444.816,173.772,19.307,153.294
C03462=1081.071,-64.534,444.805,173.773,19.309,153.294
C03463=1081.076,-64.285,444.793,173.774,19.311,153.294
C03464=1081.082,-64.035,444.781,173.776,19.312,153.294
C03465=1081.088,-63.786,444.771,173.777,19.314,153.294
C03466=1081.095,-63.536,444.759,173.779,19.315,153.294
C03467=1081.100,-63.286,444.748,173.780,19.317,153.294
C03468=1081.106,-63.036,444.736,173.782,19.319,153.294
C03469=1081.112,-62.787,444.724,173.784,19.321,153.294
C03470=1081.118,-62.537,444.713,173.785,19.322,153.294
C03471=1081.124,-62.287,444.702,173.787,19.324,153.294
C03472=1081.131,-62.038,444.690,173.788,19.325,153.294
C03473=1081.136,-61.788,444.679,173.789,19.327,153.295
C03474=1081.141,-61.539,444.668,173.791,19.329,153.295
C03475=1081.148,-61.289,444.656,173.792,19.330,153.295
C03476=1081.154,-61.039,444.645,173.794,19.332,153.295
C03477=1081.160,-60.790,444.633,173.795,19.333,153.295
C03478=1081.165,-60.540,444.622,173.797,19.335,153.295
C03479=1081.172,-60.290,444.610,173.798,19.337,153.295
C03480=1081.178,-60.041,444.599,173.799,19.338,153.295
C03481=1081.184,-59.791,444.587,173.801,19.340,153.295
C03482=1081.190,-59.541,444.575,173.802,19.342,153.295
C03483=1081.196,-59.291,444.564,173.804,19.343,153.295
C03484=1081.202,-59.042,444.552,173.805,19.345,153.295
C03485=1081.208,-58.792,444.541,173.807,19.347,153.295
C03486=1081.215,-58.542,444.530,173.809,19.348,153.295
C03487=1081.220,-58.293,444.518,173.810,19.351,153.295
C03488=1081.226,-58.043,444.507,173.812,19.352,153.296
C03489=1081.232,-57.794,444.495,173.813,19.354,153.296
C03490=1081.239,-57.544,444.484,173.814,19.355,153.296
C03491=1081.244,-57.295,444.472,173.816,19.357,153.296
C03492=1081.250,-57.044,444.460,173.817,19.359,153.296
C03493=1081.257,-56.795,444.448,173.819,19.360,153.296
C03494=1081.262,-56.545,444.437,173.820,19.362,153.296
C03495=1081.269,-56.295,444.425,173.821,19.364,153.296
C03496=1081.274,-56.046,444.414,173.823,19.365,153.296
C03497=1081.281,-55.796,444.402,173.824,19.367,153.296
C03498=1081.286,-55.547,444.391,173.827,19.369,153.296
C03499=1081.293,-55.297,444.379,173.828,19.371,153.296
C03500=1081.299,-55.047,444.367,173.829,19.372,153.296
C03501=1081.304,-54.798,444.355,173.831,19.374,153.296
C03502=1081.311,-54.548,444.343,173.832,19.376,153.296
C03503=1081.317,-54.299,444.332,173.833,19.377,153.296
C03504=1081.323,-54.049,444.320,173.835,19.379,153.297
C03505=1081.329,-53.799,444.309,173.836,19.380,153.297
C03506=1081.335,-53.550,444.297,173.838,19.382,153.297
C03507=1081.342,-53.300,444.285,173.839,19.384,153.297
C03508=1081.347,-53.050,444.273,173.841,19.385,153.297
C03509=1081.353,-52.801,444.262,173.842,19.387,153.297
C03510=1081.360,-52.551,444.250,173.844,19.389,153.297
C03511=1081.365,-52.301,444.238,173.846,19.391,153.297
C03512=1081.371,-52.052,444.226,173.847,19.392,153.297
C03513=1081.378,-51.802,444.215,173.848,19.394,153.297
C03514=1081.383,-51.552,444.203,173.850,19.396,153.297
C03515=1081.390,-51.303,444.191,173.851,19.397,153.297
C03516=1081.396,-51.053,444.180,173.852,19.399,153.297
C03517=1081.401,-50.803,444.167,173.854,19.401,153.297
C03518=1081.408,-50.554,444.155,173.855,19.402,153.297
C03519=1081.415,-50.304,444.143,173.857,19.404,153.298
C03520=1081.420,-50.055,444.132,173.858,19.406,153.298
C03521=1081.426,-49.805,444.120,173.860,19.408,153.298
C03522=1081.432,-49.532,444.106,173.862,19.410,153.298
C03523=1081.439,-49.257,444.094,173.863,19.412,153.298
C03524=1081.445,-48.984,444.080,173.865,19.414,153.298
C03525=1081.452,-48.711,444.067,173.866,19.416,153.298
C03526=1081.458,-48.461,444.055,173.868,19.417,153.298
C03527=1081.463,-48.212,444.044,173.869,19.420,153.298
C03528=1081.469,-47.962,444.031,173.870,19.421,153.298
C03529=1081.476,-47.712,444.019,173.872,19.423,153.299
C03530=1081.481,-47.463,444.007,173.873,19.425,153.299
C03531=1081.487,-47.213,443.995,173.874,19.427,153.299
C03532=1081.493,-46.963,443.983,173.877,19.429,153.299
C03533=1081.499,-46.714,443.971,173.878,19.431,153.299
C03534=1081.505,-46.464,443.959,173.879,19.432,153.299
C03535=1081.511,-46.214,443.947,173.881,19.434,153.299
C03536=1081.516,-45.965,443.935,173.882,19.436,153.299
C03537=1081.523,-45.715,443.923,173.884,19.437,153.299
C03538=1081.528,-45.466,443.911,173.885,19.439,153.299
C03539=1081.535,-45.216,443.899,173.886,19.441,153.299
C03540=1081.541,-44.966,443.887,173.888,19.443,153.300
C03541=1081.546,-44.717,443.875,173.890,19.445,153.300
C03542=1081.552,-44.467,443.863,173.891,19.447,153.300
C03543=1081.558,-44.217,443.851,173.893,19.448,153.300
C03544=1081.564,-43.967,443.838,173.894,19.450,153.300
C03545=1081.570,-43.718,443.827,173.895,19.452,153.300
C03546=1081.576,-43.468,443.814,173.896,19.454,153.300
C03547=1081.582,-43.219,443.801,173.898,19.455,153.300
C03548=1081.588,-42.970,443.790,173.900,19.458,153.300
C03549=1081.594,-42.719,443.778,173.901,19.459,153.300
C03550=1081.600,-42.470,443.766,173.903,19.461,153.300
C03551=1081.606,-42.220,443.754,173.904,19.463,153.301
C03552=1081.612,-41.971,443.741,173.905,19.465,153.301
C03553=1081.618,-41.721,443.729,173.907,19.466,153.301
C03554=1081.624,-41.471,443.717,173.908,19.468,153.301
C03555=1081.629,-41.222,443.705,173.910,19.470,153.301
C03556=1081.636,-40.972,443.693,173.912,19.472,153.301
C03557=1081.642,-40.722,443.680,173.913,19.474,153.301
C03558=1081.648,-40.473,443.668,173.914,19.476,153.301
C03559=1081.653,-40.223,443.655,173.916,19.477,153.301
C03560=1081.660,-39.974,443.643,173.917,19.479,153.301
C03561=1081.666,-39.724,443.631,173.919,19.481,153.302
C03562=1081.672,-39.474,443.618,173.920,19.483,153.302
C03563=1081.678,-39.225,443.607,173.921,19.485,153.302
C03564=1081.684,-38.975,443.594,173.923,19.487,153.302
C03565=1081.690,-38.725,443.582,173.925,19.489,153.302
C03566=1081.696,-38.476,443.570,173.926,19.491,153.302
C03567=1081.701,-38.227,443.557,173.927,19.493,153.302
C03568=1081.707,-37.977,443.545,173.929,19.494,153.302
C03569=1081.713,-37.727,443.532,173.930,19.496,153.302
C03570=1081.719,-37.477,443.520,173.931,19.498,153.303
C03571=1081.725,-37.228,443.508,173.934,19.500,153.303
C03572=1081.730,-36.978,443.495,173.935,19.502,153.303
C03573=1081.737,-36.728,443.483,173.936,19.504,153.303
C03574=1081.743,-36.478,443.470,173.937,19.506,153.303
C03575=1081.748,-36.229,443.458,173.939,19.508,153.303
C03576=1081.754,-35.979,443.446,173.940,19.509,153.303
C03577=1081.760,-35.730,443.433,173.941,19.511,153.303
C03578=1081.766,-35.480,443.420,173.943,19.514,153.303
C03579=1081.772,-35.231,443.408,173.945,19.515,153.304
C03580=1081.778,-34.981,443.395,173.946,19.517,153.304
C03581=1081.783,-34.731,443.383,173.947,19.519,153.304
C03582=1081.790,-34.482,443.371,173.949,19.521,153.304
C03583=1081.795,-34.233,443.358,173.950,19.523,153.304
C03584=1081.801,-33.983,443.346,173.952,19.525,153.304
C03585=1081.807,-33.733,443.333,173.954,19.527,153.304
C03586=1081.813,-33.460,443.319,173.955,19.529,153.304
C03587=1081.821,-33.186,443.306,173.956,19.531,153.305
C03588=1081.827,-32.914,443.292,173.958,19.533,153.305
C03589=1081.833,-32.640,443.278,173.960,19.535,153.305
C03590=1081.839,-32.391,443.265,173.961,19.537,153.305
C03591=1081.845,-32.141,443.252,173.962,19.539,153.305
C03592=1081.851,-31.892,443.240,173.964,19.541,153.305
C03593=1081.857,-31.642,443.228,173.966,19.543,153.305
C03594=1081.863,-31.392,443.215,173.967,19.545,153.305
C03595=1081.869,-31.143,443.203,173.968,19.546,153.305
C03596=1081.875,-30.894,443.190,173.970,19.548,153.306
C03597=1081.881,-30.644,443.177,173.971,19.550,153.306
C03598=1081.887,-30.394,443.165,173.973,19.552,153.306
C03599=1081.892,-30.144,443.152,173.974,19.555,153.306
C03600=1081.899,-29.895,443.139,173.976,19.556,153.306
C03601=1081.905,-29.645,443.126,173.977,19.558,153.306
C03602=1081.910,-29.396,443.114,173.978,19.560,153.306
C03603=1081.916,-29.146,443.101,173.980,19.562,153.306
C03604=1081.922,-28.896,443.088,173.982,19.564,153.306
C03605=1081.928,-28.647,443.076,173.983,19.566,153.307
C03606=1081.934,-28.397,443.063,173.985,19.568,153.307
C03607=1081.940,-28.147,443.050,173.986,19.570,153.307
C03608=1081.946,-27.897,443.037,173.987,19.572,153.307
C03609=1081.952,-27.648,443.025,173.989,19.573,153.307
C03610=1081.958,-27.398,443.011,173.991,19.576,153.307
C03611=1081.963,-27.149,442.999,173.992,19.578,153.307
C03612=1081.969,-26.899,442.987,173.993,19.579,153.307
C03613=1081.976,-26.650,442.973,173.995,19.581,153.308
C03614=1081.981,-26.400,442.961,173.996,19.583,153.308
C03615=1081.987,-26.150,442.948,173.997,19.585,153.308
C03616=1081.994,-25.901,442.935,173.999,19.587,153.308
C03617=1081.999,-25.651,442.922,174.001,19.589,153.308
C03618=1082.005,-25.402,442.909,174.002,19.591,153.308
C03619=1082.010,-25.152,442.896,174.003,19.593,153.308
C03620=1082.016,-24.902,442.884,174.005,19.595,153.308
C03621=1082.022,-24.653,442.871,174.007,19.597,153.309
C03622=1082.028,-24.403,442.858,174.008,19.599,153.309
C03623=1082.034,-24.154,442.845,174.009,19.601,153.309
C03624=1082.040,-23.904,442.832,174.011,19.603,153.309
C03625=1082.046,-23.655,442.818,174.012,19.605,153.309
C03626=1082.052,-23.405,442.806,174.013,19.607,153.309
C03627=1082.058,-23.155,442.793,174.015,19.609,153.309
C03628=1082.064,-22.906,442.780,174.016,19.611,153.310
C03629=1082.069,-22.656,442.768,174.018,19.613,153.310
C03630=1082.075,-22.407,442.754,174.019,19.615,153.310
C03631=1082.081,-22.157,442.741,174.020,19.617,153.310
